// TwinCAT 3 PLC project ExternControl
// ProgramVersion: 3.1.4024.0
// libraries:
//   Tc2_Standard, * (Beckhoff Automation GmbH)
//   Tc2_System, * (Beckhoff Automation GmbH)
//   Tc2_Utilities, * (Beckhoff Automation GmbH)
//   Tc3_Module, * (Beckhoff Automation GmbH)
//   VisuDialogs, * (System)
// project tree:
//   / GlobalTextList.TcGTLO, MAIN.TcPOU, PlcTask.TcTTO
//   MAPPING/ MAP_OUT.TcPOU (not stored), MAP_IN.TcPOU
//   MAPPING/types/ U_MOVER_CTRL.TcDUT (not stored), U_STATION_CTRL.TcDUT, U_STATION_STATE.TcDUT (not stored), U_XTS_TRANSPORT_CTRL.TcDUT, U_XTS_TRANSPORT_STATE.TcDUT (not stored)
//   PROCESS/ fb_Process.TcPOU, GVL_PROCESS.TcGVL (not stored), I_ExternControl_Process.TcIO, PROCESS_CONSTANTS.TcGVL
//   PROCESS/proc/ fb_Worker.TcPOU
//   PROCESS/_types/ E_PROCESS_TYPE.TcDUT
//   PROCESS/_Visualization/ T_PROCESS_VISU.TcVIS, PROCESS_CONTROL.TcVIS (not stored), T_XPU_VISU.TcVIS (not stored), PROCESS_XTS_TRANSPORT.TcVIS
//   XTS_TRANSPORT/CaGroup/types/ E_CA_GROUP_STATE.TcDUT (not stored), E_GROUP_CHECK.TcDUT (not stored), ST_GROUP_INFO.TcDUT
//   XTS_TRANSPORT/ GVL_XTS.TcGVL (not stored), XTS_Parameter.TcGVL
//   XTS_TRANSPORT/Mover/types/ E_MOVER_CTRL.TcDUT, E_MOVER_STATE.TcDUT, ST_GEAR_DATA.TcDUT, ST_MOVER_CTRL.TcDUT (not stored), ST_MOVER_INFO.TcDUT (not stored), ST_MOVER_STATE.TcDUT, ST_MOVE_DATA.TcDUT
//   XTS_TRANSPORT/Xpu/types/ E_XPU_CHECK.TcDUT (not stored), E_XPU_CTRL.TcDUT (not stored), E_XPU_INIT.TcDUT (not stored), E_XPU_STATE.TcDUT, ST_XPU_CTRL.TcDUT (not stored), ST_XPU_INFO.TcDUT, ST_XPU_STATE.TcDUT
//   XTS_TRANSPORT/XtsStation/_types/ E_STATION_CTRL.TcDUT (not stored), E_STATION_STATE.TcDUT (not stored), ST_STATION_CTRL.TcDUT (not stored), ST_STATION_PARAMETER.TcDUT, ST_STATION_STATE.TcDUT
//   XTS_TRANSPORT/XtsTransport/types/ E_XTS_TRANSPORT_CHECK.TcDUT (not stored), E_XTS_TRANSPORT_CTRL.TcDUT, E_XTS_TRANSPORT_STATE.TcDUT, ST_XTS_TRANSPORT_CTRL.TcDUT, ST_XTS_TRANSPORT_STATE.TcDUT (not stored)
//   XTS_TRANSPORT/_types/ E_PROGRESS.TcDUT, f_GetProgress.TcPOU, f_GetState.TcPOU (not stored), f_MoverIdDetectionModeToString.TcPOU (not stored), f_MoverPositionAssignementToString.TcPOU (not stored), f_XpuOperationModeToString.TcPOU (not stored)
//   XTS_TRANSPORT/_Visualization/ GROUP_VISU.TcVIS, STATION_VISU.TcVIS (not stored), Visualization Manager.TcVMO (not stored), XPU_VISU.TcVIS (not stored), XTS_TRANSPORT.TcVIS (not stored)
//   XTS_TRANSPORT/_Visualization/textlists/ TL_E_CTRL_STATION.TcTLO, TL_E_CTRL_TRANSPORT.TcTLO (not stored), TL_E_CTRL_XPU.TcTLO

CONFIGURATION ExternControl
    RESOURCE PLC ON TwinCAT3
        TASK PlcTask(INTERVAL := T#4ms, PRIORITY := 15);
        PROGRAM MAP_IN WITH PlcTask : MAP_IN;
        PROGRAM MAIN WITH PlcTask : MAIN;
        PROGRAM MAP_OUT WITH PlcTask : MAP_OUT;
    END_RESOURCE
END_CONFIGURATION

// ---- MAPPING/types/U_STATION_CTRL.TcDUT
{attribute 'pack_mode' := '2'}
TYPE U_STATION_CTRL :
UNION  
  _st           : ARRAY[1..MAX_STATION] OF ST_STATION_CTRL;
  _by   AT %Q*  : ARRAY[1..MAX_STATION] OF
                  ARRAY[1..SIZEOF(ST_STATION_CTRL)] OF BYTE;
END_UNION
END_TYPE

// ---- MAPPING/types/U_XTS_TRANSPORT_CTRL.TcDUT
{attribute 'pack_mode' := '2'}
TYPE U_XTS_TRANSPORT_CTRL :
UNION
  _st           : ST_XTS_TRANSPORT_CTRL;
  _by   AT%Q*   : ARRAY[1..SIZEOF(ST_XTS_TRANSPORT_CTRL)] OF BYTE;
END_UNION
END_TYPE

// ---- PROCESS/_types/E_PROCESS_TYPE.TcDUT
{attribute 'qualified_only'}
{attribute 'strict'}
{attribute 'to_string'}
TYPE E_PROCESS_TYPE :
(
	NULL,             // nothing happens here
  SINGLE,           // single XTS Station
  PARALLEL,         // synced station handshakes for multiple XTS Stations, same process on all stations, all who enter are processed
  PARALLEL_STRICT,  // synced station handshakes for multiple XTS Stations, same process on all stations, all who are enabled must be processed
  SERIAL,           // synced station handshakes for multiple XTS Stations, all mover have to go through all stations in process
  DISTRIBUTOR       // single XTS Station, no work done here, automated distribution for LastTarget to FirstTarget
)UINT;
END_TYPE

// ---- XTS_TRANSPORT/CaGroup/types/ST_GROUP_INFO.TcDUT
TYPE ST_GROUP_INFO :
STRUCT
  GroupStatusValid,
  GroupStatusBusy,
  GroupMoving, 
  GroupHoming, 
  GroupErrorStop, 
  GroupNotReady, 
  GroupStandby, 
  GroupStopping,
 
  GroupDisabled, 
  AllAxesStanding, 
  ConstantVelocity, 
  Accelerating, 
  Decelerating, 
  InPosition, 
  GroupError					  : BIT; 

  GroupErrorId					: UDINT;

  AxisCount      				: UDINT;
  AxisCountEnabled      : UDINT;

  {attribute 'displaymode':='hex'}
  CaGroupOID            : OTCID;

  CaGroupState          : E_CA_GROUP_STATE;
END_STRUCT
END_TYPE

// ---- XTS_TRANSPORT/Mover/types/E_MOVER_CTRL.TcDUT
{attribute 'qualified_only'}
{attribute 'strict'}
{attribute 'to_string'}
TYPE E_MOVER_CTRL :
(
  MOVER_NULL,               // initial value at startup, used for change of order or retrigger
  MOVER_ENABLE,             // sets MC_Power.Enable
  MOVER_DISABLE,            // removes MC_Power.Enable
  MOVER_MOVE_TO_POS,        // modulo absolute positioning with MC_MoveAbsolute, InTargetPosition check
  MOVER_MOVE_TO_POS_CA,     // modulo absolute positioning with MC_MoveAbsoluteCA, InTargetPosition check
  MOVER_SEND_TO_POS_CA,     // modulo absolute positioning with MC_MoveAbsoluteCA, done after moving ReleaseDistance
  MOVER_HALT,               // halts mover; by use of MC_Halt mover is set passive in CA group
  MOVER_GEAR_IN,            // GearIn for mover in standstill

  MOVER_GEAR_IN_POS_CA,     // GearInPosCA of mover; when FB_GearInPosCa is InSync --> order is done; check SyncDistance yourself and release mover with e_mover_order.mover_SendToPos
  MOVER_GEAR_OUT,           // gear out for mover
  MOVER_RESET               // MC_RESET for mover
)UINT;
END_TYPE

// ---- XTS_TRANSPORT/Mover/types/E_MOVER_STATE.TcDUT
{attribute 'qualified_only'}
{attribute 'to_string'}
TYPE E_MOVER_STATE :
(
  MOVER_NULL,               // initial value at startup, used for change of order or retrigger
  MOVER_ENABLE,             // sets MC_Power.Enable
  MOVER_DISABLE,            // removes MC_Power.Enable
  MOVER_MOVE_TO_POS,        // modulo absolute positioning with MC_MoveAbsolute, InTargetPosition check
  MOVER_MOVE_TO_POS_CA,     // modulo absolute positioning with MC_MoveAbsoluteCA, InTargetPosition check
  MOVER_SEND_TO_POS_CA,     // modulo absolute positioning with MC_MoveAbsoluteCA, done after moving ReleaseDistance
  MOVER_HALT,               // halts mover; by use of MC_Halt mover is set passive in CA group
  MOVER_GEAR_IN,            // GearIn for mover in standstill

  MOVER_GEAR_IN_POS_CA,     // GearInPosCA of mover; when FB_GearInPosCa is InSync --> order is done; check SyncDistance yourself and release mover with e_mover_order.mover_SendToPos
  MOVER_GEAR_OUT,           // gear out for mover
  MOVER_RESET               // MC_RESET for mover
)UINT;
END_TYPE

// ---- XTS_TRANSPORT/Mover/types/ST_GEAR_DATA.TcDUT
{attribute 'pack_mode' := '2'}
TYPE ST_GEAR_DATA :
STRUCT
  rDeltaToMasterPos       : REAL;
  rModuloSyncPosSlave     : REAL;
  rMasterStartDistance    : REAL;
  rGearNumerator          : REAL;
  iGearDenumerator        : USINT  := 1;
END_STRUCT
END_TYPE

// ---- XTS_TRANSPORT/Mover/types/ST_MOVER_STATE.TcDUT
{attribute 'pack_mode' := '2'}
TYPE ST_MOVER_STATE :
STRUCT
  State           : E_MOVER_STATE;  // ST_MOVER_CTRL.Cmd with added E_PROGRESS
  MasterId        : USINT;            // mirror NC AxisId of Master axis
END_STRUCT
END_TYPE

// ---- XTS_TRANSPORT/Mover/types/ST_MOVE_DATA.TcDUT
{attribute 'pack_mode' := '2'}
TYPE ST_MOVE_DATA :
STRUCT
  // HAUD 2024 03 14
  // some init data added for example
  rPos            : LREAL :=   2275.0;
  rVelo           : LREAL :=    500.0;
  rAcc            : LREAL :=   5000.0;
  rJerk           : LREAL := 500000.0;
  rGap            : LREAL :=    100.0;
  rOverride       : LREAL :=    100.0;
  rDelta          : LREAL :=      0.05;
  rDistance       : LREAL :=     25.0;
END_STRUCT
END_TYPE

// ---- XTS_TRANSPORT/Xpu/types/E_XPU_STATE.TcDUT
{attribute 'to_string'}
TYPE E_XPU_STATE :
(
  XTS_NULL,
  XTS_INVALID,
  XTS_INIT                      := 10,    // initialize XPU
  XTS_STATION_INFO_READ         := 20,    // get Station information from Xpu
  XTS_IDLE                      := 30
)UINT;
END_TYPE

// ---- XTS_TRANSPORT/Xpu/types/ST_XPU_INFO.TcDUT
{attribute 'pack_mode' := '2'}
TYPE ST_XPU_INFO :
STRUCT
  AllPositionsValid   : BIT;
  IdDetectionError    : BIT;
  IdDetectionValid    : BIT;
  IdDetectionActive   : BIT;

  OperationMode       : UINT;

  IdDetectionMode           : UINT;
  MoverPositionAssignement  : UINT;

  nDetectedAxisCount  : UINT;
  nExpectedAxisCount  : UINT;

  
END_STRUCT
END_TYPE

// ---- XTS_TRANSPORT/Xpu/types/ST_XPU_STATE.TcDUT
{attribute 'pack_mode' := '2'}
TYPE ST_XPU_STATE :
STRUCT
  Init            : E_XPU_INIT;
  State           : E_XPU_STATE;
  Check           : E_XPU_CHECK;
  DcLink          : BIT;
END_STRUCT
END_TYPE

// ---- XTS_TRANSPORT/XtsStation/_types/ST_STATION_PARAMETER.TcDUT
TYPE ST_STATION_PARAMETER :
STRUCT
  sText             : STRING(80); // only description
  rPosWait          : REAL;       // start of station, a sending station is using this value to send mover to
  rReleaseDistance  : REAL;       // distance from stop pos mover has to travel (from ActPos) in order for station to go back to mover detection

  rGap              : REAL;
  rVelo             : REAL;
  rAccDec           : REAL;
  rJerk             : REAL;

  // how many nests (stop positions) mover has to stop at (1 = default)
  nConfiguredStopCount  : USINT := 1; // 1-8 --> NestMask = BYTE

  // mover stop position in station, relative to rPosWait!!
  rPosStop          : ARRAY[1..8] OF LREAL;
END_STRUCT
END_TYPE

// ---- XTS_TRANSPORT/XtsStation/_types/ST_STATION_STATE.TcDUT
{attribute 'pack_mode' := '2'}
TYPE ST_STATION_STATE :
STRUCT
  eState          : E_STATION_STATE;
  {attribute 'displaymode':='bin'}
  nMask           : BYTE;
  nMoverId        : USINT;
  rMoverModPos    : lreal; // modulo position of detected mover
  nQueue          : USINT; // queue count for station
END_STRUCT
END_TYPE

// ---- XTS_TRANSPORT/XtsTransport/types/E_XTS_TRANSPORT_CTRL.TcDUT
{attribute 'strict'}
{attribute 'to_string'}
TYPE E_XTS_TRANSPORT_CTRL :
(
  CMD_NULL,
  CMD_INIT                  := 10,  // Xpu, Group, Mover initialization: clear errors, clear group, check Xpu data, check mover detection
  CMD_IDLE,

  CMD_MOVER_ENABLE          := 20,  // all mover are enabled, checked for ControlLoopClosed
  CMD_MOVER_DISABLE,                // all mover are disabled, no axis in CaGroup: no error, any axis in CaGroup: group error

  CMD_GROUP_CLEAR           := 30,  // halt all movers, clear errors, remove all movers from group, clear group
  CMD_GROUP_BUILD,                  // add all movers to group
  CMD_GROUP_ENABLE,                 // group with movers is enabled

  CMD_TRANSPORT_START       := 40,  // move all mover[i] to start position
  CMD_TRANSPORT_RESTART             // move all mover[i] to LastPosition[i]

)UINT;
END_TYPE

// ---- XTS_TRANSPORT/XtsTransport/types/E_XTS_TRANSPORT_STATE.TcDUT
{attribute 'to_string'}
TYPE E_XTS_TRANSPORT_STATE :
(
  TRANSPORT_NULL,
  TRANSPORT_INVALID,
  TRANSPORT_INIT            := 10,  // Xpu, Group, Mover initialization: init TcCOM objects, clear errors, clear group, check Xpu data, check mover detection
  TRANSPORT_IDLE,                   // cyclic check for errors, check Xpu data

  TRANSPORT_MOVER_ENABLE    := 20,  // all mover are enabled, checked for ControlLoopClosed
  TRANSPORT_MOVER_DISABLE,          // all mover are disabled

  TRANSPORT_GROUP_CLEAR     := 30,  // halt all movers, clear errors, remove all movers from group, clear group
  TRANSPORT_GROUP_BUILD,            // add all movers to group
  TRANSPORT_GROUP_ENABLE,           // group with movers is enabled

  TRANSPORT_START           := 40,  // move all mover[i] to start position
  TRANSPORT_RESTART                 // move all mover[i] to LastPosition[i]
)UINT;
END_TYPE

// ---- XTS_TRANSPORT/XtsTransport/types/ST_XTS_TRANSPORT_CTRL.TcDUT
TYPE ST_XTS_TRANSPORT_CTRL :
STRUCT
  Cmd       : E_XTS_TRANSPORT_CTRL;
END_STRUCT
END_TYPE

// ---- XTS_TRANSPORT/_types/E_PROGRESS.TcDUT
{attribute 'qualified_only'}
{attribute 'to_string'}
TYPE E_PROGRESS :
(
  PROGRESS_INVALID,
  PROGRESS_INIT           :=  1000,
  PROGRESS_BUSY           :=  2000,
  PROGRESS_PREPARE        :=  3000,
  PROGRESS_STARTUP        :=  4000,
  PROGRESS_CHECK          :=  5000,
  PROGRESS_OCCUPIED       :=  6000,
  PROGRESS_WORKING        :=  7000,
  PROGRESS_STILL_WORKING  :=  8000,
  PROGRESS_ERROR          :=  9000,
  PROGRESS_DONE           := 10000
)UINT;
END_TYPE

// ---- PROCESS/PROCESS_CONSTANTS.TcGVL
//{attribute 'qualified_only'}
VAR_GLOBAL CONSTANT
  MAX_PROCESS       : UINT := 9;

  DISTRIBUTOR_2     : UINT := 9;// 9
  DISTRIBUTOR_1     : UINT := 8;// 8
  OUTPUT_R2         : UINT := 7;// 7
  OUTPUT_R1         : UINT := 6;// 6
  BUFFER_3          : UINT := 5;// 5
  OUTPUT_1          : UINT := 4;// 4
  INPUT             : UINT := 3;// 3
  BUFFER_1          : UINT := 2;// 2
  BUFFER_4          : UINT := 1;// 1

  QUEUE_COUNT       : UINT := 12; // 
END_VAR

// ---- XTS_TRANSPORT/XTS_Parameter.TcGVL
//{attribute 'qualified_only'}
VAR_GLOBAL CONSTANT
// HAUD 2024 04 30 - introduction of fb_UnitControl
  Version             : STRING  := '3.2.8';

  MAX_MOVER           : UINT    := 96;

  MAX_STATION         : UINT    := 53;
  MAX_STATION_NEST    : UINT    := TO_UINT(SIZEOF(ST_STATION_STATE.nMask)*8);

END_VAR

// ---- PROCESS/I_ExternControl_Process.TcIO
INTERFACE I_ExternControl_Process

METHOD PUBLIC DelBitWord : WORD
VAR_INPUT
  inVal   : WORD;
  bitNo   : DINT;
END_VAR
END_METHOD

PROPERTY EnableProcess : word
GET
END_GET
SET
END_SET
END_PROPERTY

METHOD PUBLIC GetBitDWord : BOOL
VAR_INPUT
  inVal   : DWORD;
  bitNo   : DINT;
END_VAR
END_METHOD

METHOD PUBLIC GetBitWord : BOOL
VAR_INPUT
  inVal   : WORD;
  bitNo   : DINT;
END_VAR
END_METHOD

METHOD PUBLIC Init : BOOL
END_METHOD

PROPERTY MoverCountInQueue : uint
GET
END_GET
END_PROPERTY

PROPERTY MoverInQueue : Bool
GET
END_GET
END_PROPERTY

PROPERTY ProcessCmd : E_STATION_CTRL
SET
END_SET
END_PROPERTY

PROPERTY ProcessPerMinute : uint
GET
END_GET
END_PROPERTY

PROPERTY ProcessState : E_STATION_STATE
GET
END_GET
END_PROPERTY

PROPERTY ProcessType : e_process_type
GET
END_GET
SET
END_SET
END_PROPERTY

METHOD PUBLIC SetBitDWord : DWORD
VAR_INPUT
  inVal   : DWORD;
  bitNo   : DINT;
END_VAR
END_METHOD

METHOD PUBLIC SetBitWord : WORD
VAR_INPUT
  inVal   : WORD;
  bitNo   : DINT;
END_VAR
END_METHOD

PROPERTY StationCount : uint
GET
END_GET
END_PROPERTY

PROPERTY StationFirst : uint
GET
END_GET
SET
END_SET
END_PROPERTY

PROPERTY TargetMask : dword
GET
END_GET
SET
END_SET
END_PROPERTY

END_INTERFACE

// ---- MAPPING/MAP_IN.TcPOU
PROGRAM MAP_IN
VAR

  {attribute 'TcLinkTo' := '._by := TIPC^XtsTransport^XtsTransport Instance^PlcTask Outputs^MAP_OUT.uTransportState._by'}
  uTransportState     : U_XTS_TRANSPORT_STATE;
  {attribute 'TcLinkTo' := '._by := TIPC^XtsTransport^XtsTransport Instance^PlcTask Outputs^MAP_OUT.uStationState._by'}
  uStationState       : U_STATION_STATE;
END_VAR

          // destination address
                                            // source address
                                                                    // size
  memcpy(ADR(GVL_XTS.XtsTransportState),  ADR(uTransportState),   SIZEOF(ST_XTS_TRANSPORT_STATE));
  memcpy(ADR(GVL_XTS.StationState),       ADR(uStationState),     SIZEOF(uStationState));

END_PROGRAM

// ---- MAIN.TcPOU
//---------------------------------------------------------------------------------------------------------------
//
//  HAUD 2024.04.13
//
//  - ExternControl for XtsTransport
//
//  - example project for controlling XTS transport layer
//  - transport layer members:
//
//      HAUD 2024 04 30 - introduction of fb_UnitControl as interface to APPLICATION
//
//    - fb_UnitControl
//      - groups commands into sequences for APPLICATION
//      - handles XtsTransport
//      - handles fb_Process
//
//    - fb_Process
//      - groups XtsStations for processes
//      - synced handshakes with all assigned XtsStations
//
//    - Transport Control Unit
//      - mapped from XtsTransport GVL_XTS.TransportCtrl / GVL_XTS.TransportState
//        - Info for CaGroup
//        - Info for Xpu
//
//      - coordinates members to get XTS in defined states
//
//    - Xts Stations
//      - handshakes for mover transport
//
//---------------------------------------------------------------------------------------------------------------
// This SOFTWARE is provided as an Exemple by THE PROVIDER "as is" and "with all faults." THE PROVIDER makes no 
// representations or warranties of any kind concerning the safety, suitability, lack of viruses, inaccuracies, 
// typographical errors, or other harmful components of this SOFTWARE. There are inherent dangers in the use of 
// any software, and you are solely responsible for determining whether this SOFTWARE is compatible with your 
// equipment and other software installed on your equipment. You are also solely responsible for the protection 
// of your equipment and backup of your data, and THE PROVIDER will not be liable for any damages you may suffer 
// in connection with using, modifying, or distributing this SOFTWARE.
//---------------------------------------------------------------------------------------------------------------
PROGRAM MAIN
VAR
  bInit,
  bStart              : BOOL;
  eInit               : E_PROGRESS;

  nProcess,
  nStation            : UINT;

  tProcess            : ARRAY[1..MAX_PROCESS] OF TIME;

  {attribute 'displaymode':='bin'}
  wEnableProcess      : ARRAY[1..MAX_PROCESS] OF DWORD;  // switch XTS stations on/off here (one word per process --> max. 16 stations each)

  {attribute 'displaymode':='bin'}
  wInitProcess        : WORD;  // processes init

  bEmptySerialStation : BOOL;

  eProcessCmd         : ARRAY[1..MAX_PROCESS] OF E_STATION_CTRL;
  eProcessState       : ARRAY[1..MAX_PROCESS] OF E_STATION_STATE;

  nMoverSelected,
  nStationSelected,
  nProcessSelected,
  nStationParameter   : UINT;

  eTransportCmd,
  eTransportCmdOld    : E_XTS_TRANSPORT_CTRL;

  eTransportState,
  eTransportStateOld  : E_XTS_TRANSPORT_STATE;
  eTransportResult,
  eStateStart         : E_PROGRESS;

  eXpuState           : E_XPU_STATE;
  eXpuResult          : E_PROGRESS;
  eXpuCheck           : E_XPU_CHECK;

  eMoverState         : E_MOVER_STATE;
  eMoverResult        : E_PROGRESS;

  sCaGroupState,
  sTransportState,
  sTransportCheck,
  sTransportResult,
  sXpuState,
  sXpuResult,
  sXpuCheck,
  sXpuOpMode,
  sXpuMoverdetectionMode,
  sXpuMoverAssignement,
  sMoverState,
  sMoverResult,
  sStationState,
  sStationStateMask,
  sStationCtrlMask,
  sProcessEnableMask        : STRING;

  bStationEnable,
  bStationEnter,
  bStationStart,
  bStationDone,
  bStationOut,
  bStationGone            : BOOL;

  sStationText            : STRING;
  nVariant                : uint;
END_VAR

//#############################################################################
// Visualization data	
//#############################################################################	
VisuData();
//
//#############################################################################
// check for changed Cmd on XtsTransportCtrl.Cmd
//#############################################################################
//
eTransportCmd                         := GVL_XTS.XtsTransportCtrl.Cmd;
//
IF (eTransportCmd <> eTransportCmdOld)
THEN
  eTransportCmdOld                    := eTransportCmd;
  bStart                              := FALSE;
  bEmptySerialStation                 := FALSE;
  eStateStart                         := E_PROGRESS.PROGRESS_INIT;
  memset(ADR(wEnableProcess), 0, SIZEOF(wEnableProcess));

  CASE eTransportCmd
  OF
    E_XTS_TRANSPORT_CTRL.CMD_INIT:
      bInit                           := FALSE;

  ELSE
    IF bInit
    THEN
      CASE eTransportCmd
      OF
        E_XTS_TRANSPORT_CTRL.CMD_IDLE,
        E_XTS_TRANSPORT_CTRL.CMD_TRANSPORT_START:
          FOR nProcess := 1 TO MAX_PROCESS
          DO
            eProcessCmd[nProcess]     := E_STATION_CTRL.STATION_DISABLE;
          END_FOR
      END_CASE
    END_IF
  END_CASE
END_IF
//
//
//#############################################################################
// check for changed state on XtsTransportState.State
//#############################################################################
//
IF (GVL_XTS.XtsTransportState.State <> eTransportStateOld)
THEN
  CASE (GVL_XTS.XtsTransportState.State MOD E_PROGRESS.PROGRESS_DONE)
  OF
    E_XTS_TRANSPORT_STATE.TRANSPORT_START:
      CASE eStateStart
      OF
        E_PROGRESS.PROGRESS_INIT:
          IF GVL_XTS.XtsTransportState.GroupInfo.AllAxesStanding
          THEN
            eStateStart               := E_PROGRESS.PROGRESS_BUSY;
            memset(ADR(wEnableProcess), 0, SIZEOF(wEnableProcess));
          END_IF

        E_PROGRESS.PROGRESS_BUSY:
          eStateStart                   := E_PROGRESS.PROGRESS_PREPARE;
          FOR nProcess := 1 TO MAX_PROCESS
          DO
            FOR nStation := 1 TO GVL_PROCESS.Process[nProcess].StationCount
            DO
              wEnableProcess[nProcess]  := GVL_PROCESS.Process[nProcess].SetBitDWord(wEnableProcess[nProcess],(nStation-1));
            END_FOR
            //wEnableProcess[OUTPUT_R1] := 1;
            GVL_PROCESS.Process[nProcess].EnableProcess := TO_WORD(wEnableProcess[nProcess]);
          END_FOR
          FOR nProcess := 1 TO MAX_PROCESS
          DO
            IF (nProcess = MAX_PROCESS)
            THEN
              GVL_PROCESS.Process[nProcess].TargetMask := wEnableProcess[1];
            ELSE
              GVL_PROCESS.Process[nProcess].TargetMask := wEnableProcess[nProcess+1];
            END_IF
          END_FOR
          FOR nStation := 0 TO (GVL_PROCESS.Process[BUFFER_3].TargetLast - GVL_PROCESS.Process[BUFFER_3].TargetFirst)
          DO 
            GVL_PROCESS.Process[BUFFER_3].TargetMask     := GVL_PROCESS.Process[BUFFER_3].SetBitDWord(GVL_PROCESS.Process[BUFFER_3].TargetMask,(nStation));
          END_FOR

        E_PROGRESS.PROGRESS_PREPARE:
          eStateStart                 := E_PROGRESS.PROGRESS_STARTUP;
          FOR nProcess := 1 TO MAX_PROCESS
          DO
            IF NOT (GVL_PROCESS.Process[nProcess].EnableProcess = wEnableProcess[nProcess])
            THEN
              eStateStart             := E_PROGRESS.PROGRESS_PREPARE;
            END_IF
          END_FOR

        E_PROGRESS.PROGRESS_STARTUP:
          eTransportStateOld          := GVL_XTS.XtsTransportState.State;
          bStart                      := TRUE;
      END_CASE

  ELSE
    eTransportStateOld                := GVL_XTS.XtsTransportState.State;

    CASE (GVL_XTS.XtsTransportState.State MOD E_PROGRESS.PROGRESS_ERROR)
    OF
      E_XTS_TRANSPORT_STATE.TRANSPORT_START:
        bStart                        := FALSE;

    END_CASE
  END_CASE
END_IF
//
//#############################################################################
//#############################################################################
//
IF NOT bInit
THEN
  Init();
  ProcessConfig_2x12_DST_02();
END_IF
//#############################################################################
//#############################################################################
// cyclic call to processes
//#############################################################################
FOR nProcess := 1 TO MAX_PROCESS
DO
  GVL_PROCESS.Process[nProcess].Cycle();

  GVL_PROCESS.Process[nProcess].EnabledStation    := ADR(GVL_PROCESS.StationsEnabled);  // enabled process: for other processes to read
  GVL_PROCESS.Process[nProcess].MoverPerMinute    := ADR(GVL_PROCESS.MoverPerMinute);

  GVL_PROCESS.Process[nProcess].StationCtrl       := ADR(GVL_XTS.StationCtrl);
  GVL_PROCESS.Process[nProcess].StationState      := ADR(GVL_XTS.StationState);

  GVL_PROCESS.ItfProcess[nProcess]                := GVL_PROCESS.Process[nProcess]; 
END_FOR


//#############################################################################
// process workers
//#############################################################################
GVL_PROCESS.Distributor2.ProcessTime    := tProcess[DISTRIBUTOR_2];
GVL_PROCESS.Distributor2.ProcessIndex   := DISTRIBUTOR_2;
GVL_PROCESS.Distributor2.ItfProcesses   REF= GVL_PROCESS.ItfProcess;

GVL_PROCESS.Distributor1.ProcessTime    := tProcess[DISTRIBUTOR_1];
GVL_PROCESS.Distributor1.ProcessIndex   := DISTRIBUTOR_1;
GVL_PROCESS.Distributor1.ItfProcesses   REF= GVL_PROCESS.ItfProcess;

GVL_PROCESS.OutputR2.ProcessTime        := tProcess[OUTPUT_R2];
GVL_PROCESS.OutputR2.ProcessIndex       := OUTPUT_R2;
GVL_PROCESS.OutputR2.ItfProcesses       REF= GVL_PROCESS.ItfProcess;

GVL_PROCESS.OutputR1.ProcessTime        := tProcess[OUTPUT_R1];
GVL_PROCESS.OutputR1.ProcessIndex       := OUTPUT_R1;
GVL_PROCESS.OutputR1.ItfProcesses       REF= GVL_PROCESS.ItfProcess;

GVL_PROCESS.Buffer3.ProcessTime         := tProcess[BUFFER_3];
GVL_PROCESS.Buffer3.ProcessIndex        := BUFFER_3;
GVL_PROCESS.Buffer3.ItfProcesses        REF= GVL_PROCESS.ItfProcess;

GVL_PROCESS.Output1.ProcessTime         := tProcess[OUTPUT_1];
GVL_PROCESS.Output1.ProcessIndex        := OUTPUT_1;
GVL_PROCESS.Output1.ItfProcesses        REF= GVL_PROCESS.ItfProcess;

GVL_PROCESS.Input1.ProcessTime          := tProcess[INPUT];
GVL_PROCESS.Input1.ProcessIndex         := INPUT;
GVL_PROCESS.Input1.ItfProcesses         REF= GVL_PROCESS.ItfProcess;

GVL_PROCESS.Buffer1.ProcessTime         := tProcess[BUFFER_1];
GVL_PROCESS.Buffer1.ProcessIndex        := BUFFER_1;
GVL_PROCESS.Buffer1.ItfProcesses        REF= GVL_PROCESS.ItfProcess;

GVL_PROCESS.Buffer1.ProcessTime         := tProcess[BUFFER_1];
GVL_PROCESS.Buffer4.ProcessIndex        := BUFFER_4;
GVL_PROCESS.Buffer4.ItfProcesses        REF= GVL_PROCESS.ItfProcess;

//#############################################################################
//
IF NOT (bInit) THEN RETURN; END_IF
//
//#############################################################################
//#############################################################################

IF (nVariant = 0)
THEN
  GVL_PROCESS.Distributor2.AUTO(bStart);
  GVL_PROCESS.Distributor1.AUTO(bStart);
  GVL_PROCESS.OutputR2.AUTO(bStart);
  GVL_PROCESS.OutputR1.AUTO(bStart);
  GVL_PROCESS.Buffer3.AUTO(bStart);
  GVL_PROCESS.Output1.AUTO(bStart);
  GVL_PROCESS.Input1.AUTO(bStart);
  GVL_PROCESS.Buffer1.AUTO(bStart);
  GVL_PROCESS.Buffer4.AUTO(bStart);

ELSIF (nVariant = 1)
THEN
  GVL_PROCESS.Distributor2.AUTO_1(bStart);
  GVL_PROCESS.Distributor1.AUTO_1(bStart);
  GVL_PROCESS.OutputR2.AUTO_1(bStart);
  GVL_PROCESS.OutputR1.AUTO_1(bStart);
  GVL_PROCESS.Buffer3.AUTO_1(bStart);
  GVL_PROCESS.Output1.AUTO_1(bStart);
  GVL_PROCESS.Input1.AUTO_1(bStart);
  GVL_PROCESS.Buffer1.AUTO_1(bStart);
  GVL_PROCESS.Buffer4.AUTO_1(bStart);
END_IF















//#############################################################################

METHOD Init
VAR_INPUT
END_VAR
CASE eInit
OF
  E_PROGRESS.PROGRESS_INVALID,
  E_PROGRESS.PROGRESS_DONE:
    bStart                          := FALSE;
    eInit                           := E_PROGRESS.PROGRESS_INIT;
    GVL_XTS.XtsTransportCtrl.Cmd    := E_XTS_TRANSPORT_CTRL.CMD_NULL;

  E_PROGRESS.PROGRESS_INIT:
    IF (GVL_XTS.XtsTransportState.XpuInfo.IdDetectionValid) OR
       (GVL_XTS.XtsTransportState.XpuInfo.OperationMode = 1) // Simulation
    THEN
      GVL_XTS.XtsTransportCtrl.Cmd  := E_XTS_TRANSPORT_CTRL.CMD_INIT;

      IF (GVL_xts.XtsTransportState.State = E_XTS_TRANSPORT_STATE.TRANSPORT_INIT + E_PROGRESS.PROGRESS_DONE)
      THEN
        GVL_XTS.XtsTransportCtrl.Cmd:= E_XTS_TRANSPORT_CTRL.CMD_IDLE;
        eInit                       := E_PROGRESS.PROGRESS_BUSY;
      END_IF
    END_IF

  E_PROGRESS.PROGRESS_BUSY:
    eInit                           := E_PROGRESS.PROGRESS_PREPARE;
    wInitProcess                    := 0;
    ProcessConfig_1x12();
    ProcessConfig_2x12();

  E_PROGRESS.PROGRESS_PREPARE:
    ProcessConfig_2x12_DST_02();

    FOR nProcess := 1 TO MAX_PROCESS
    DO
      GVL_PROCESS.Process[nProcess].ProcessCmd         := E_STATION_CTRL.STATION_INIT;
      IF (GVL_PROCESS.Process[nProcess].ProcessState = E_STATION_STATE.STATION_INIT)
      THEN
        wInitProcess                := GVL_PROCESS.Process[nProcess].SetBitWord(wInitProcess,  (nProcess-1));
      END_IF
    END_FOR
    IF (wInitProcess = EXPT(2,MAX_PROCESS)-1)
    THEN
      eInit                         := E_PROGRESS.PROGRESS_STARTUP;
    END_IF

  E_PROGRESS.PROGRESS_STARTUP:
    StationParameterInit();

    tProcess[INPUT]                 := T#450MS;
    tProcess[OUTPUT_1]              := T#600MS;
    tProcess[OUTPUT_R1]             := T#600MS;
    tProcess[OUTPUT_R2]             := T#600MS;

    FOR nProcess := 1 TO MAX_PROCESS
    DO
      GVL_PROCESS.Process[nProcess].ProcessCmd         := E_STATION_CTRL.STATION_DISABLE;
    END_FOR
    bInit                           := TRUE;
    eInit                           := E_PROGRESS.PROGRESS_DONE;

END_CASE
END_METHOD

METHOD ProcessConfig_1x12
VAR
  _nProcess     : UINT;
END_VAR

      // BUFFER_4
      _nProcess                       := 1;
      GVL_PROCESS.Process[_nProcess].ProcessType   := E_PROCESS_TYPE.DISTRIBUTOR;
      GVL_PROCESS.Process[_nProcess].StationFirst  := 52;
      GVL_PROCESS.Process[_nProcess].StationLast   := 52;
      GVL_PROCESS.Process[_nProcess].TargetFirst   := 53;
      GVL_PROCESS.Process[_nProcess].TargetLast    := 53;

      // BUFFER_1
      _nProcess                       := 2;
      GVL_PROCESS.Process[_nProcess].ProcessType   := E_PROCESS_TYPE.DISTRIBUTOR;
      GVL_PROCESS.Process[_nProcess].StationFirst  := 53;
      GVL_PROCESS.Process[_nProcess].StationLast   := 53;
      GVL_PROCESS.Process[_nProcess].TargetFirst   :=  1;
      GVL_PROCESS.Process[_nProcess].TargetLast    := 12;

      // INPUT
      _nProcess                       := 3;
      tProcess[_nProcess]             := T#850MS;
      GVL_PROCESS.Process[_nProcess].ProcessType   := E_PROCESS_TYPE.PARALLEL;
      GVL_PROCESS.Process[_nProcess].StationFirst  :=  1;
      GVL_PROCESS.Process[_nProcess].StationLast   := 12;
      GVL_PROCESS.Process[_nProcess].TargetFirst   := 13;
      GVL_PROCESS.Process[_nProcess].TargetLast    := 24;

      // OUTPUT_1
      _nProcess                       := 4;
      tProcess[_nProcess]             := T#850MS;
      GVL_PROCESS.Process[_nProcess].ProcessType   := E_PROCESS_TYPE.PARALLEL;
      GVL_PROCESS.Process[_nProcess].StationFirst  := 13;
      GVL_PROCESS.Process[_nProcess].StationLast   := 24;
      GVL_PROCESS.Process[_nProcess].TargetFirst   := 50;
      GVL_PROCESS.Process[_nProcess].TargetLast    := 50;

      // DISTRIBUTOR_1
      _nProcess                        := 8;
      GVL_PROCESS.Process[_nProcess].ProcessType   := E_PROCESS_TYPE.DISTRIBUTOR;
      GVL_PROCESS.Process[_nProcess].StationFirst  := 50;
      GVL_PROCESS.Process[_nProcess].StationLast   := 50;
      GVL_PROCESS.Process[_nProcess].TargetFirst   := 51;
      GVL_PROCESS.Process[_nProcess].TargetLast    := 51;

      // DISTRIBUTOR_2
      _nProcess                        := 9;
      GVL_PROCESS.Process[_nProcess].ProcessType   := E_PROCESS_TYPE.DISTRIBUTOR;
      GVL_PROCESS.Process[_nProcess].StationFirst  := 51;
      GVL_PROCESS.Process[_nProcess].StationLast   := 51;
      GVL_PROCESS.Process[_nProcess].TargetFirst   := 52;
      GVL_PROCESS.Process[_nProcess].TargetLast    := 52;
END_METHOD

METHOD ProcessConfig_2x12
VAR
  _nProcess     : UINT;
END_VAR
    
      // BUFFER_4
      _nProcess                       := BUFFER_4;
      GVL_PROCESS.Process[_nProcess].ProcessType   := E_PROCESS_TYPE.DISTRIBUTOR;
      GVL_PROCESS.Process[_nProcess].StationFirst  := 52;
      GVL_PROCESS.Process[_nProcess].StationLast   := 52;
      GVL_PROCESS.Process[_nProcess].TargetFirst   := 53;
      GVL_PROCESS.Process[_nProcess].TargetLast    := 53;

      // BUFFER_1
      _nProcess                       := BUFFER_1;
      GVL_PROCESS.Process[_nProcess].ProcessType   := E_PROCESS_TYPE.DISTRIBUTOR;
      GVL_PROCESS.Process[_nProcess].StationFirst  := 53;
      GVL_PROCESS.Process[_nProcess].StationLast   := 53;
      GVL_PROCESS.Process[_nProcess].TargetFirst   :=  1;
      GVL_PROCESS.Process[_nProcess].TargetLast    := 12;

      // INPUT
      _nProcess                       := INPUT;
      GVL_PROCESS.Process[_nProcess].ProcessType   := E_PROCESS_TYPE.PARALLEL;
      GVL_PROCESS.Process[_nProcess].StationFirst  :=  1;
      GVL_PROCESS.Process[_nProcess].StationLast   := 12;
      GVL_PROCESS.Process[_nProcess].TargetFirst   := 25;
      GVL_PROCESS.Process[_nProcess].TargetLast    := 25;

      // BUFFER_3
      _nProcess                        := BUFFER_3;
      GVL_PROCESS.Process[_nProcess].ProcessType   := E_PROCESS_TYPE.DISTRIBUTOR;
      GVL_PROCESS.Process[_nProcess].StationFirst  := 25;
      GVL_PROCESS.Process[_nProcess].StationLast   := 25;
      GVL_PROCESS.Process[_nProcess].TargetFirst   := 26;
      GVL_PROCESS.Process[_nProcess].TargetLast    := 49;

      // OUTPUT_R1
      _nProcess                        := OUTPUT_R1;
      GVL_PROCESS.Process[_nProcess].ProcessType   := E_PROCESS_TYPE.PARALLEL_STRICT;
      GVL_PROCESS.Process[_nProcess].StationFirst  := 26;
      GVL_PROCESS.Process[_nProcess].StationLast   := 37;
      GVL_PROCESS.Process[_nProcess].TargetFirst   := 50;
      GVL_PROCESS.Process[_nProcess].TargetLast    := 50;

      // OUTPUT_R2
      _nProcess                        := OUTPUT_R2;
      GVL_PROCESS.Process[_nProcess].ProcessType   := E_PROCESS_TYPE.PARALLEL_STRICT;
      GVL_PROCESS.Process[_nProcess].StationFirst  := 38;
      GVL_PROCESS.Process[_nProcess].StationLast   := 49;
      GVL_PROCESS.Process[_nProcess].TargetFirst   := 50;
      GVL_PROCESS.Process[_nProcess].TargetLast    := 50;

      // DISTRIBUTOR_1
      _nProcess                        := DISTRIBUTOR_1;
      GVL_PROCESS.Process[_nProcess].ProcessType   := E_PROCESS_TYPE.DISTRIBUTOR;
      GVL_PROCESS.Process[_nProcess].StationFirst  := 50;
      GVL_PROCESS.Process[_nProcess].StationLast   := 50;
      GVL_PROCESS.Process[_nProcess].TargetFirst   := 51;
      GVL_PROCESS.Process[_nProcess].TargetLast    := 51;

      // DISTRIBUTOR_2
      _nProcess                        := DISTRIBUTOR_2;
      GVL_PROCESS.Process[_nProcess].ProcessType   := E_PROCESS_TYPE.DISTRIBUTOR;
      GVL_PROCESS.Process[_nProcess].StationFirst  := 51;
      GVL_PROCESS.Process[_nProcess].StationLast   := 51;
      GVL_PROCESS.Process[_nProcess].TargetFirst   := 52;
      GVL_PROCESS.Process[_nProcess].TargetLast    := 52;
END_METHOD

METHOD ProcessConfig_2x12_DST_02
VAR
  _nProcess     : UINT;
END_VAR
    
      // BUFFER_4
      _nProcess                       := BUFFER_4;
      GVL_PROCESS.Process[_nProcess].ProcessType   := E_PROCESS_TYPE.DISTRIBUTOR;
      GVL_PROCESS.Process[_nProcess].StationFirst  := 52;
      GVL_PROCESS.Process[_nProcess].StationLast   := 52;
      GVL_PROCESS.Process[_nProcess].TargetFirst   := 53;
      GVL_PROCESS.Process[_nProcess].TargetLast    := 53;

      // BUFFER_1
      _nProcess                       := BUFFER_1;
      GVL_PROCESS.Process[_nProcess].ProcessType   := E_PROCESS_TYPE.DISTRIBUTOR;
      GVL_PROCESS.Process[_nProcess].StationFirst  := 53;
      GVL_PROCESS.Process[_nProcess].StationLast   := 53;
      GVL_PROCESS.Process[_nProcess].TargetFirst   :=  1;
      GVL_PROCESS.Process[_nProcess].TargetLast    := 12;

      // INPUT
      _nProcess                       := INPUT;
      GVL_PROCESS.Process[_nProcess].ProcessType   := E_PROCESS_TYPE.PARALLEL;
      GVL_PROCESS.Process[_nProcess].StationFirst  :=  1;
      GVL_PROCESS.Process[_nProcess].StationLast   := 12;
      GVL_PROCESS.Process[_nProcess].TargetFirst   := 25;
      GVL_PROCESS.Process[_nProcess].TargetLast    := 25;

      // BUFFER_3
      _nProcess                        := BUFFER_3;
      GVL_PROCESS.Process[_nProcess].ProcessType   := E_PROCESS_TYPE.DISTRIBUTOR;
      GVL_PROCESS.Process[_nProcess].StationFirst  := 25;
      GVL_PROCESS.Process[_nProcess].StationLast   := 25;
      GVL_PROCESS.Process[_nProcess].TargetFirst   := 26;
      GVL_PROCESS.Process[_nProcess].TargetLast    := 49;

      // OUTPUT_R1
      _nProcess                        := OUTPUT_R1;
      GVL_PROCESS.Process[_nProcess].ProcessType   := E_PROCESS_TYPE.PARALLEL_STRICT;
      GVL_PROCESS.Process[_nProcess].StationFirst  := 26;
      GVL_PROCESS.Process[_nProcess].StationLast   := 37;
      GVL_PROCESS.Process[_nProcess].TargetFirst   := 51;
      GVL_PROCESS.Process[_nProcess].TargetLast    := 51;

      // OUTPUT_R2
      _nProcess                        := OUTPUT_R2;
      GVL_PROCESS.Process[_nProcess].ProcessType   := E_PROCESS_TYPE.PARALLEL_STRICT;
      GVL_PROCESS.Process[_nProcess].StationFirst  := 38;
      GVL_PROCESS.Process[_nProcess].StationLast   := 49;
      GVL_PROCESS.Process[_nProcess].TargetFirst   := 51;
      GVL_PROCESS.Process[_nProcess].TargetLast    := 51;

      // DISTRIBUTOR_1
      _nProcess                        := DISTRIBUTOR_1;
      GVL_PROCESS.Process[_nProcess].ProcessType   := E_PROCESS_TYPE.DISTRIBUTOR;
      GVL_PROCESS.Process[_nProcess].StationFirst  := 50;
      GVL_PROCESS.Process[_nProcess].StationLast   := 50;
      GVL_PROCESS.Process[_nProcess].TargetFirst   := 51;
      GVL_PROCESS.Process[_nProcess].TargetLast    := 51;

      // DISTRIBUTOR_2
      _nProcess                        := DISTRIBUTOR_2;
      GVL_PROCESS.Process[_nProcess].ProcessType   := E_PROCESS_TYPE.DISTRIBUTOR;
      GVL_PROCESS.Process[_nProcess].StationFirst  := 51;
      GVL_PROCESS.Process[_nProcess].StationLast   := 51;
      GVL_PROCESS.Process[_nProcess].TargetFirst   := 52;
      GVL_PROCESS.Process[_nProcess].TargetLast    := 52;
END_METHOD

ACTION StationParameterInit:
//-----------------------------------------------------------------------------
//
//  HAUD 2024.06.12
//
// 
//  - hard coded station parameter
//-----------------------------------------------------------------------------
//-----------------------------------------------------------------------------

//-----------------------------------------------------------------------------------------------------------------------------------------
//  INPUT
    sStationText  := 'INPUT';
//-----------------------------------------------------------------------------------------------------------------------------------------
nStationParameter := 1;
GVL_XTS.StationParameter[nStationParameter].sText                 := sStationText;
GVL_XTS.StationParameter[nStationParameter].rPosWait              :=    988.0;  // absolute modulo position


//-----------------------------------------------------------------------------------------------------------------------------------------
nStationParameter := 2;
GVL_XTS.StationParameter[nStationParameter].sText                 := sStationText;
GVL_XTS.StationParameter[nStationParameter].rPosWait              :=    988.0; // absolute modulo position


//-----------------------------------------------------------------------------------------------------------------------------------------
nStationParameter := 3;
GVL_XTS.StationParameter[nStationParameter].sText                 := sStationText;
GVL_XTS.StationParameter[nStationParameter].rPosWait              :=    988.0; // absolute modulo position


//-----------------------------------------------------------------------------------------------------------------------------------------
nStationParameter := 4;
GVL_XTS.StationParameter[nStationParameter].sText                 := sStationText;
GVL_XTS.StationParameter[nStationParameter].rPosWait              :=   988.0;  // absolute modulo position


//-----------------------------------------------------------------------------------------------------------------------------------------
nStationParameter := 5;
GVL_XTS.StationParameter[nStationParameter].sText                 := sStationText;
GVL_XTS.StationParameter[nStationParameter].rPosWait              :=   988.0;  // absolute modulo position


//-----------------------------------------------------------------------------------------------------------------------------------------
nStationParameter := 6;
GVL_XTS.StationParameter[nStationParameter].sText                 := sStationText;
GVL_XTS.StationParameter[nStationParameter].rPosWait              :=   988.0;  // absolute modulo position


//-----------------------------------------------------------------------------------------------------------------------------------------
nStationParameter := 7;
GVL_XTS.StationParameter[nStationParameter].sText                 := sStationText;
GVL_XTS.StationParameter[nStationParameter].rPosWait              :=   988.0;  // absolute modulo position


//-----------------------------------------------------------------------------------------------------------------------------------------
nStationParameter := 8;
GVL_XTS.StationParameter[nStationParameter].sText                 := sStationText;
GVL_XTS.StationParameter[nStationParameter].rPosWait              :=   988.0;  // absolute modulo position


//-----------------------------------------------------------------------------------------------------------------------------------------
nStationParameter := 9;
GVL_XTS.StationParameter[nStationParameter].sText                 := sStationText;
GVL_XTS.StationParameter[nStationParameter].rPosWait              :=   988.0;  // absolute modulo position


//-----------------------------------------------------------------------------------------------------------------------------------------
nStationParameter := 10;
GVL_XTS.StationParameter[nStationParameter].sText                 := sStationText;
GVL_XTS.StationParameter[nStationParameter].rPosWait              :=   988.0;  // absolute modulo position


//-----------------------------------------------------------------------------------------------------------------------------------------
nStationParameter := 11;
GVL_XTS.StationParameter[nStationParameter].sText                 := sStationText;
GVL_XTS.StationParameter[nStationParameter].rPosWait              :=   988.0;  // absolute modulo position


//-----------------------------------------------------------------------------------------------------------------------------------------
nStationParameter := 12;
GVL_XTS.StationParameter[nStationParameter].sText                 := sStationText;
GVL_XTS.StationParameter[nStationParameter].rPosWait              :=   988.0;  // absolute modulo position


//-----------------------------------------------------------------------------------------------------------------------------------------
//-----------------------------------------------------------------------------------------------------------------------------------------
//  OUTPUT_1
    sStationText  := 'OUTPUT_1';
//-----------------------------------------------------------------------------------------------------------------------------------------
nStationParameter := 13;
GVL_XTS.StationParameter[nStationParameter].sText                 := sStationText;
GVL_XTS.StationParameter[nStationParameter].rPosWait              :=   3582.0;  // absolute modulo position


//-----------------------------------------------------------------------------------------------------------------------------------------
nStationParameter := 14;
GVL_XTS.StationParameter[nStationParameter].sText                 := sStationText;
GVL_XTS.StationParameter[nStationParameter].rPosWait              :=   3582.0;  // absolute modulo position


//-----------------------------------------------------------------------------------------------------------------------------------------
nStationParameter := 15;
GVL_XTS.StationParameter[nStationParameter].sText                 := sStationText;
GVL_XTS.StationParameter[nStationParameter].rPosWait              :=   3582.0;  // absolute modulo position


//-----------------------------------------------------------------------------------------------------------------------------------------
nStationParameter := 16;
GVL_XTS.StationParameter[nStationParameter].sText                 := sStationText;
GVL_XTS.StationParameter[nStationParameter].rPosWait              :=   3582.0;  // absolute modulo position


//-----------------------------------------------------------------------------------------------------------------------------------------
nStationParameter := 17;
GVL_XTS.StationParameter[nStationParameter].sText                 := sStationText;
GVL_XTS.StationParameter[nStationParameter].rPosWait              :=   3582.0;  // absolute modulo position


//-----------------------------------------------------------------------------------------------------------------------------------------
nStationParameter := 18;
GVL_XTS.StationParameter[nStationParameter].sText                 := sStationText;
GVL_XTS.StationParameter[nStationParameter].rPosWait              :=   3582.0;  // absolute modulo position


//-----------------------------------------------------------------------------------------------------------------------------------------
nStationParameter := 19;
GVL_XTS.StationParameter[nStationParameter].sText                 := sStationText;
GVL_XTS.StationParameter[nStationParameter].rPosWait              :=   3582.0;  // absolute modulo position


//-----------------------------------------------------------------------------------------------------------------------------------------
nStationParameter := 20;
GVL_XTS.StationParameter[nStationParameter].sText                 := sStationText;
GVL_XTS.StationParameter[nStationParameter].rPosWait              :=   3582.0;  // absolute modulo position


//-----------------------------------------------------------------------------------------------------------------------------------------
nStationParameter := 21;
GVL_XTS.StationParameter[nStationParameter].sText                 := sStationText;
GVL_XTS.StationParameter[nStationParameter].rPosWait              :=   3582.0;  // absolute modulo position


//-----------------------------------------------------------------------------------------------------------------------------------------
nStationParameter := 22;
GVL_XTS.StationParameter[nStationParameter].sText                 := sStationText;
GVL_XTS.StationParameter[nStationParameter].rPosWait              :=   3582.0;  // absolute modulo position


//-----------------------------------------------------------------------------------------------------------------------------------------
nStationParameter := 23;
GVL_XTS.StationParameter[nStationParameter].sText                 := sStationText;
GVL_XTS.StationParameter[nStationParameter].rPosWait              :=   3582.0;  // absolute modulo position


//-----------------------------------------------------------------------------------------------------------------------------------------
nStationParameter := 24;
GVL_XTS.StationParameter[nStationParameter].sText                 := sStationText;
GVL_XTS.StationParameter[nStationParameter].rPosWait              :=   3582.0;  // absolute modulo position


//-----------------------------------------------------------------------------------------------------------------------------------------
//-----------------------------------------------------------------------------------------------------------------------------------------
//  BUFFER_3
    sStationText  := 'BUFFER_3';
//-----------------------------------------------------------------------------------------------------------------------------------------
nStationParameter := 25;
GVL_XTS.StationParameter[nStationParameter].sText                 := sStationText;
GVL_XTS.StationParameter[nStationParameter].rPosWait              :=   6000.0;  // absolute modulo position


//-----------------------------------------------------------------------------------------------------------------------------------------
//-----------------------------------------------------------------------------------------------------------------------------------------
//  OUTPUT_R1
    sStationText  := 'OUTPUT_R1';
//-----------------------------------------------------------------------------------------------------------------------------------------
nStationParameter := 26;
GVL_XTS.StationParameter[nStationParameter].sText                 := sStationText;
GVL_XTS.StationParameter[nStationParameter].rPosWait              :=   7000.0;  // absolute modulo position


//-----------------------------------------------------------------------------------------------------------------------------------------
nStationParameter := 27;
GVL_XTS.StationParameter[nStationParameter].sText                 := sStationText;
GVL_XTS.StationParameter[nStationParameter].rPosWait              :=   7000.0;  // absolute modulo position


//-----------------------------------------------------------------------------------------------------------------------------------------
nStationParameter := 28;
GVL_XTS.StationParameter[nStationParameter].sText                 := sStationText;
GVL_XTS.StationParameter[nStationParameter].rPosWait              :=   7000.0;  // absolute modulo position


//-----------------------------------------------------------------------------------------------------------------------------------------
nStationParameter := 29;
GVL_XTS.StationParameter[nStationParameter].sText                 := sStationText;
GVL_XTS.StationParameter[nStationParameter].rPosWait              :=   7000.0;  // absolute modulo position


//-----------------------------------------------------------------------------------------------------------------------------------------
nStationParameter := 30;
GVL_XTS.StationParameter[nStationParameter].sText                 := sStationText;
GVL_XTS.StationParameter[nStationParameter].rPosWait              :=   7000.0;  // absolute modulo position


//-----------------------------------------------------------------------------------------------------------------------------------------
nStationParameter := 31;
GVL_XTS.StationParameter[nStationParameter].sText                 := sStationText;
GVL_XTS.StationParameter[nStationParameter].rPosWait              :=   7000.0;  // absolute modulo position


//-----------------------------------------------------------------------------------------------------------------------------------------
nStationParameter := 32;
GVL_XTS.StationParameter[nStationParameter].sText                 := sStationText;
GVL_XTS.StationParameter[nStationParameter].rPosWait              :=   7000.0;  // absolute modulo position


//-----------------------------------------------------------------------------------------------------------------------------------------
nStationParameter := 33;
GVL_XTS.StationParameter[nStationParameter].sText                 := sStationText;
GVL_XTS.StationParameter[nStationParameter].rPosWait              :=   7000.0;  // absolute modulo position


//-----------------------------------------------------------------------------------------------------------------------------------------
nStationParameter := 34;
GVL_XTS.StationParameter[nStationParameter].sText                 := sStationText;
GVL_XTS.StationParameter[nStationParameter].rPosWait              :=   7000.0;  // absolute modulo position


//-----------------------------------------------------------------------------------------------------------------------------------------
nStationParameter := 35;
GVL_XTS.StationParameter[nStationParameter].sText                 := sStationText;
GVL_XTS.StationParameter[nStationParameter].rPosWait              :=   7000.0;  // absolute modulo position


//-----------------------------------------------------------------------------------------------------------------------------------------
nStationParameter := 36;
GVL_XTS.StationParameter[nStationParameter].sText                 := sStationText;
GVL_XTS.StationParameter[nStationParameter].rPosWait              :=   7000.0;  // absolute modulo position


//-----------------------------------------------------------------------------------------------------------------------------------------
nStationParameter := 37;
GVL_XTS.StationParameter[nStationParameter].sText                 := sStationText;
GVL_XTS.StationParameter[nStationParameter].rPosWait              :=   7000.0;  // absolute modulo position


//-----------------------------------------------------------------------------------------------------------------------------------------
//-----------------------------------------------------------------------------------------------------------------------------------------
//  OUTPUT_R2
    sStationText  := 'OUTPUT_R2';
//-----------------------------------------------------------------------------------------------------------------------------------------
nStationParameter := 38;
GVL_XTS.StationParameter[nStationParameter].sText                 := sStationText;
GVL_XTS.StationParameter[nStationParameter].rPosWait              :=   7000.0;  // absolute modulo position


//-----------------------------------------------------------------------------------------------------------------------------------------
nStationParameter := 39;
GVL_XTS.StationParameter[nStationParameter].sText                 := sStationText;
GVL_XTS.StationParameter[nStationParameter].rPosWait              :=   7000.0;  // absolute modulo position


//-----------------------------------------------------------------------------------------------------------------------------------------
nStationParameter := 40;
GVL_XTS.StationParameter[nStationParameter].sText                 := sStationText;
GVL_XTS.StationParameter[nStationParameter].rPosWait              :=   7000.0;  // absolute modulo position


//-----------------------------------------------------------------------------------------------------------------------------------------
nStationParameter := 41;
GVL_XTS.StationParameter[nStationParameter].sText                 := sStationText;
GVL_XTS.StationParameter[nStationParameter].rPosWait              :=   7000.0;  // absolute modulo position


//-----------------------------------------------------------------------------------------------------------------------------------------
nStationParameter := 42;
GVL_XTS.StationParameter[nStationParameter].sText                 := sStationText;
GVL_XTS.StationParameter[nStationParameter].rPosWait              :=   7000.0;  // absolute modulo position


//-----------------------------------------------------------------------------------------------------------------------------------------
nStationParameter := 43;
GVL_XTS.StationParameter[nStationParameter].sText                 := sStationText;
GVL_XTS.StationParameter[nStationParameter].rPosWait              :=   7000.0;  // absolute modulo position


//-----------------------------------------------------------------------------------------------------------------------------------------
nStationParameter := 44;
GVL_XTS.StationParameter[nStationParameter].sText                 := sStationText;
GVL_XTS.StationParameter[nStationParameter].rPosWait              :=   7000.0;  // absolute modulo position


//-----------------------------------------------------------------------------------------------------------------------------------------
nStationParameter := 45;
GVL_XTS.StationParameter[nStationParameter].sText                 := sStationText;
GVL_XTS.StationParameter[nStationParameter].rPosWait              :=   7000.0;  // absolute modulo position


//-----------------------------------------------------------------------------------------------------------------------------------------
nStationParameter := 46;
GVL_XTS.StationParameter[nStationParameter].sText                 := sStationText;
GVL_XTS.StationParameter[nStationParameter].rPosWait              :=   7000.0;  // absolute modulo position


//-----------------------------------------------------------------------------------------------------------------------------------------
nStationParameter := 47;
GVL_XTS.StationParameter[nStationParameter].sText                 := sStationText;
GVL_XTS.StationParameter[nStationParameter].rPosWait              :=   7000.0;  // absolute modulo position


//-----------------------------------------------------------------------------------------------------------------------------------------
nStationParameter := 48;
GVL_XTS.StationParameter[nStationParameter].sText                 := sStationText;
GVL_XTS.StationParameter[nStationParameter].rPosWait              :=   7000.0;  // absolute modulo position


//-----------------------------------------------------------------------------------------------------------------------------------------
nStationParameter := 49;
GVL_XTS.StationParameter[nStationParameter].sText                 := sStationText;
GVL_XTS.StationParameter[nStationParameter].rPosWait              :=   7000.0;  // absolute modulo position



//-----------------------------------------------------------------------------------------------------------------------------------------
//-----------------------------------------------------------------------------------------------------------------------------------------
//  DISTRIBUTOR_1
    sStationText  := 'DISTRIBUTOR_1';
//-----------------------------------------------------------------------------------------------------------------------------------------
nStationParameter := 50;
GVL_XTS.StationParameter[nStationParameter].sText                 := sStationText;
GVL_XTS.StationParameter[nStationParameter].rPosWait              :=  10000.0;  // absolute modulo position


//-----------------------------------------------------------------------------------------------------------------------------------------
//-----------------------------------------------------------------------------------------------------------------------------------------
// DISTRIBUTOR_2
    sStationText  := 'DISTRIBUTOR_2';
//-----------------------------------------------------------------------------------------------------------------------------------------
nStationParameter := 51;
GVL_XTS.StationParameter[nStationParameter].sText                 := sStationText;
GVL_XTS.StationParameter[nStationParameter].rPosWait              :=  11500.0;  // absolute modulo position


//-----------------------------------------------------------------------------------------------------------------------------------------
//-----------------------------------------------------------------------------------------------------------------------------------------
//  BUFFER_4
    sStationText  := 'BUFFER_4';
//-----------------------------------------------------------------------------------------------------------------------------------------
nStationParameter := 52;
GVL_XTS.StationParameter[nStationParameter].sText                 := sStationText;
GVL_XTS.StationParameter[nStationParameter].rPosWait              :=  20000.0;  // absolute modulo position


//-----------------------------------------------------------------------------------------------------------------------------------------
//-----------------------------------------------------------------------------------------------------------------------------------------
//  BUFFER_1
    sStationText  := 'BUFFER_1';
//-----------------------------------------------------------------------------------------------------------------------------------------
nStationParameter := 53;
GVL_XTS.StationParameter[nStationParameter].sText                 := sStationText;
GVL_XTS.StationParameter[nStationParameter].rPosWait              :=    150.0;  // absolute modulo position
END_ACTION

METHOD VisuData
VAR_INPUT
END_VAR

// get enumerations from XPU for visu:
eTransportState                       := f_GetState   (GVL_XTS.XtsTransportState.State);
eTransportResult                      := f_GetProgress(GVL_XTS.XtsTransportState.State);

eXpuState                             := f_GetState   (GVL_XTS.XtsTransportState.XpuState.State);
eXpuResult                            := f_GetProgress(GVL_XTS.XtsTransportState.XpuState.State);

eXpuCheck                             := GVL_XTS.XtsTransportState.XpuState.Check;

// display xpu state and result in visu
// get strings and info
sCaGroupState                         := TO_STRING(GVL_XTS.XtsTransportState.GroupInfo.CaGroupState);

sTransportState                       := TO_STRING(eTransportState);
sTransportCheck                       := TO_STRING(GVL_XTS.XtsTransportState.Check);
sTransportResult                      := TO_STRING(eTransportResult);

sXpuState                             := TO_STRING(eXpuState);
sXpuResult                            := TO_STRING(eXpuResult);
sXpuCheck                             := TO_STRING(eXpuCheck);

sXpuOpMode                            := f_XpuOperationModeToString         (GVL_XTS.XtsTransportState.XpuInfo.OperationMode);
sXpuMoverdetectionMode                := f_MoverIdDetectionModeToString     (GVL_XTS.XtsTransportState.XpuInfo.IdDetectionMode);
sXpuMoverAssignement                  := f_MoverPositionAssignementToString (GVL_XTS.XtsTransportState.XpuInfo.MoverPositionAssignement);

nMoverSelected                        := SEL((nMoverSelected<1), nMoverSelected, 1);
nMoverSelected                        := SEL((nMoverSelected>MAX_MOVER), nMoverSelected, MAX_MOVER);

nStationSelected                      := SEL((nStationSelected<1), nStationSelected, 1);
nStationSelected                      := SEL((nStationSelected>MAX_STATION), nStationSelected, MAX_STATION);

nProcessSelected                      := SEL((nProcessSelected<1), nProcessSelected, 1);
nProcessSelected                      := SEL((nProcessSelected>MAX_PROCESS), nProcessSelected, MAX_PROCESS);

bStationEnable                        := SEL((GVL_XTS.StationCtrl[nStationSelected].eCmd = E_STATION_CTRL.STATION_ENABLE),        FALSE, TRUE);
bStationEnter                         := SEL((GVL_XTS.StationCtrl[nStationSelected].eCmd = E_STATION_CTRL.STATION_MOVER_ENTER),   FALSE, TRUE);
bStationStart                         := SEL((GVL_XTS.StationCtrl[nStationSelected].eCmd = E_STATION_CTRL.STATION_PROCESS_START), FALSE, TRUE);
bStationDone                          := SEL((GVL_XTS.StationCtrl[nStationSelected].eCmd = E_STATION_CTRL.STATION_PROCESS_DONE),  FALSE, TRUE);
bStationOut                           := SEL((GVL_XTS.StationCtrl[nStationSelected].eCmd = E_STATION_CTRL.STATION_MOVER_OUT),     FALSE, TRUE);
bStationGone                          := SEL((GVL_XTS.StationCtrl[nStationSelected].eCmd = E_STATION_CTRL.STATION_MOVER_GONE),    FALSE, TRUE);

sStationState                         := TO_STRING(GVL_XTS.StationState[nStationSelected].eState);
sStationStateMask                     := Tc2_Utilities.BYTE_TO_BINSTR(GVL_XTS.StationState[nStationSelected].nMask, 8);
sStationCtrlMask                      := Tc2_Utilities.BYTE_TO_BINSTR(GVL_XTS.StationCtrl[nStationSelected].nMask, 8);

sProcessEnableMask                    := Tc2_Utilities.WORD_TO_BINSTR(GVL_PROCESS.Process[nProcessSelected].EnableProcess, 16);
END_METHOD

END_PROGRAM

// ---- XTS_TRANSPORT/_types/f_GetProgress.TcPOU
// global function to extract e_progress from combined value
FUNCTION f_GetProgress : uint
VAR_INPUT
  state     : UINT;
END_VAR
VAR
  nP        : uint;
END_VAR


nP := state / E_PROGRESS.PROGRESS_INIT;

f_GetProgress := nP * E_PROGRESS.PROGRESS_INIT;

END_FUNCTION

// ---- PROCESS/fb_Process.TcPOU
//---------------------------------------------------------------------------------------------------------------
//
//  HAUD 2023.03.27
//
//  TR08
//  - XTS_TRANSPORT_LAYER
//
//  fb_Process
//  - grouping of xts stations to sync start process
//  - nFirst to nLast xts stations are checked for starting process simultaneously
//  - basic preparation of station target index in PrepareTarget()
//  - handshake with station control for mover transport through station
//
//---------------------------------------------------------------------------------------------------------------
// This SOFTWARE is provided as an Exemple by THE PROVIDER "as is" and "with all faults." THE PROVIDER makes no 
// representations or warranties of any kind concerning the safety, suitability, lack of viruses, inaccuracies, 
// typographical errors, or other harmful components of this SOFTWARE. There are inherent dangers in the use of 
// any software, and you are solely responsible for determining whether this SOFTWARE is compatible with your 
// equipment and other software installed on your equipment. You are also solely responsible for the protection 
// of your equipment and backup of your data, and THE PROVIDER will not be liable for any damages you may suffer 
// in connection with using, modifying, or distributing this SOFTWARE.
//---------------------------------------------------------------------------------------------------------------
FUNCTION_BLOCK fb_Process IMPLEMENTS I_ExternControl_Process
VAR
  _eType                      : E_PROCESS_TYPE;   // types of process: SINGLE, PARALLEL, SERIAL, DISTRIBUTOR
  _sCheck                     : STRING;

  _eProcessCmd                : E_STATION_CTRL;   // control from property
  _eProcessState              : E_STATION_STATE;  // state   to   property

  {attribute 'displaymode':='bin'}
  _wEnableProcess             : WORD; // control sets bits to switch on stations
  _bEnabledStation            : POINTER TO ARRAY[1..XTS_Parameter.MAX_STATION]  OF BOOL; // information about all enabled xts stations

  // xts stations
  _stCtrl                     : POINTER TO ARRAY[1..XTS_Parameter.MAX_STATION]  OF ST_STATION_CTRL;
  _stState                    : POINTER TO ARRAY[1..XTS_Parameter.MAX_STATION]  OF ST_STATION_STATE;

  // who is included in process
  // _nFirst to _nLast MUST be in closed consecutive order
  _nStation,
  _nStationCount,
  _nFirstStation,
  _nLastStation               : UINT;

  // work vars for writing onto _stCtrl[nStation].nTargetStation
  _nTarget,
  _nFirstTarget,
  _nLastTarget                : UINT;   // for parallel process xts stations and the last xts station in serial process

  _nSerialTarget              : ARRAY[1..XTS_Parameter.MAX_STATION]  OF UINT; // serial targets within process

  _nPreparedTarget            : ARRAY[1..XTS_Parameter.MAX_MOVER]  OF UINT;   // targets for parallel and single process

  // bitmasks for station states in CycleStation()
  {attribute 'displaymode':='bin'}
  _wEnable                    : WORD;   // commanded enable of xts station
  {attribute 'displaymode':='bin'}
  _wEnter                     : WORD;   // mover asking for entry into xts station
  {attribute 'displaymode':='bin'}
  _wStart                     : WORD;   // xts station asking for process handshake
  {attribute 'displaymode':='bin'}
  _wLeave                     : WORD;   // xts station wants to send out mover
  {attribute 'displaymode':='bin'}
  _wQueue                     : WORD;   // mover was entered into xts station list
  {attribute 'displaymode':='bin'}
  _wMoverInStation            : WORD;   // mover entry was granted, mover is now in station
  {attribute 'displaymode':='bin'}
  _wError                     : WORD;   // minor error, must be fixed by _stCtrl[nStation]
  {attribute 'displaymode':='bin'}
  _wErrorFatal                : WORD;   // fatal error, must be fixed by debugging
  {attribute 'displaymode':='bin'}
  _wTargetId                  : WORD;   // nTargetStation > 0 in _stDtrl[nStation].nTargetStation

  {attribute 'displaymode':='bin'}
  _TargetMask                 : DWORD;   // bit positions correspond to index of xts station
 
  _bNext                      : BOOL;

  _nProcessPerMinute          : uint; // sum of all xts stations output per minute in process
  _rtrigProcess               : ARRAY[1..XTS_Parameter.MAX_STATION] OF Tc2_Standard.R_TRIG;
  _tonPartsPerMinute          : Tc2_Standard.TON;

  _nMoverPerMinute            : POINTER TO ARRAY[1..XTS_Parameter.MAX_STATION]  OF UINT;
  _nMoverCount,
  _nMoverCountOld             : ARRAY[1..XTS_Parameter.MAX_STATION]  OF UINT;

  _eDistributorTarget         : E_PROGRESS;

END_VAR

METHOD private Check : BOOL

IF (_nFirstStation < 1) OR
   (_nFirstStation > MAX_STATION)
THEN
  _sCheck                     := '_nFirstStation out of bounds';
  RETURN;
END_IF

IF (_nLastStation < 1) OR
   (_nLastStation > MAX_STATION)
THEN
  _sCheck                     := '_nLastStation out of bounds';
  RETURN;
END_IF

IF (_nFirstTarget < 1) OR
   (_nFirstTarget > MAX_STATION)
THEN
  _sCheck                     := '_nFirstTarget out of bounds';
  RETURN;
END_IF

IF (_nLastTarget < 1) OR
   (_nLastTarget > MAX_STATION)
THEN
  _sCheck                     := '_nLastTarget out of bounds';
  RETURN;
END_IF

IF NOT (_stCtrl  <> 0)
THEN
  _sCheck                     := '_stCtrl: missing pointer';
  RETURN;
END_IF

IF NOT (_stState <> 0)
THEN
  _sCheck                     := '_stState: missing pointer';
  RETURN;
END_IF

IF NOT (_bEnabledStation  <> 0)
THEN
  _sCheck                     := '_bEnableStation: missing pointer';
  RETURN;
END_IF

IF not (_nMoverPerMinute <> 0)
THEN
  _sCheck                     := '_nMoverPerMinute: missing pointer';
  RETURN;
END_IF

_nStationCount                := _nLastStation - _nFirstStation + 1;

IF (_nStationCount < 1) OR
   (_nStationCount > (SIZEOF(WORD)*8))
THEN
  _sCheck                     := '_nStationCount out of bounds';
  RETURN;
END_IF


_sCheck                       := TO_STRING(E_PROGRESS.PROGRESS_DONE);
Check                         := TRUE;
END_METHOD

METHOD Cycle
VAR_INST
  _nStn     : uint;
END_VAR
IF NOT Check() THEN RETURN; END_IF


//-----------------------------------------------------------------------------
// collect state information from xts stations
// state information is collected in Masks (WORD), 
// every bit represents one XTS station in process
//-----------------------------------------------------------------------------
//  _wEnable                        : enable cmd was given to xts station
//  _wEnter                         : a mover is requesting entry
//  _wStart                         : mover has arrived and xts station is ready
//  _wLeave                         : xts station wants to send mover out
//  _wQueue                         : somebody's waiting
//  _wMoverInStation                : mover is in station
//  _wError                         : error state for handshake
//  _wErrorFatal                    : error state for severe problems (debugging required)
//  _wTargetId                      : Ctrl.nTargetStation > 0
//  _wMoverInQueueSerial            : SERIAL process: bits to check whether a mover is waiting to be processed
//
CycleStation();                     // get state information from all XtsStations in process
//-----------------------------------------------------------------------------
//-----------------------------------------------------------------------------
//  E_STATION_CTRL.STATION_INIT: hard reset of process and XtsStations
//-----------------------------------------------------------------------------
CASE _eProcessCmd                   // check input property
OF
  E_STATION_CTRL.STATION_INIT:      // commanded init from ctrl
    CASE _eType
    OF
      E_PROCESS_TYPE.SERIAL:
        InitSerialTargets();
    END_CASE
    Init();                         RETURN; // rest you will, return you must
END_CASE
//-----------------------------------------------------------------------------
// E_STATION_STATE.STATION_INIT: pass through here and switch off XtsStations
//-----------------------------------------------------------------------------
CASE _eProcessState                 // check output property
OF
  E_STATION_STATE.STATION_INIT:     // xts station empty, disabled by default
    _eProcessState                  := E_STATION_STATE.STATION_DISABLE;
    FOR _nStn := _nLastStation TO _nFirstStation BY(-1) 
    DO
      _stCtrl^[_nStn].eCmd          := E_STATION_CTRL.STATION_DISABLE;
    END_FOR

END_CASE
//-----------------------------------------------------------------------------
//  E_STATION_STATE.STATION_DISABLE: wait for enable from flow control
//-----------------------------------------------------------------------------
CASE _eProcessState                 // check output property
OF
  E_STATION_STATE.STATION_DISABLE:  // check for enable command
    IF (_eProcessCmd = E_STATION_CTRL.STATION_ENABLE)
    THEN
      _eProcessState                := E_STATION_STATE.STATION_ENABLE;

      FOR _nStn := _nLastStation TO _nFirstStation BY(-1) 
      DO
          _stCtrl^[_nStn].eCmd      := E_STATION_CTRL.STATION_ENABLE;
      END_FOR
    END_IF
END_CASE
//-----------------------------------------------------------------------------
//  E_STATION_STATE.STATION_ENABLE: check Cmd and wait for XtsStations to be enabled
//-----------------------------------------------------------------------------
CASE _eProcessState
OF
  E_STATION_STATE.STATION_ENABLE:
    CASE _eProcessCmd
    OF
      E_STATION_CTRL.STATION_DISABLE:
        _eProcessState              := E_STATION_STATE.STATION_INIT;

      E_STATION_CTRL.STATION_ENABLE:
        IF (_wEnable = _wEnableProcess)
        THEN
          InitSerialTargets();
          _eProcessState            := E_STATION_STATE.STATION_DETECT_MOVER;
        END_IF
    END_CASE
END_CASE
//-----------------------------------------------------------------------------
// E_STATION_STATE.STATION_DETECT_MOVER: wait for any XtsStation to 
//                                       have a mover ready to enter
//-----------------------------------------------------------------------------
CASE _eProcessState
OF
  E_STATION_STATE.STATION_DETECT_MOVER:
    CASE _eProcessCmd
    OF
      E_STATION_CTRL.STATION_DISABLE:
        _eProcessState              := E_STATION_STATE.STATION_INIT;

      E_STATION_CTRL.STATION_ENABLE:
        IF (_wEnter > 0)            // at least one mover is asking for entry
        THEN
          _eDistributorTarget       := E_PROGRESS.PROGRESS_INVALID;

                                    // switch process state in order to tell process control
          _eProcessState            := E_STATION_STATE.STATION_MOVER_ENTER;
        END_IF
    END_CASE
END_CASE
//-----------------------------------------------------------------------------
//  E_STATION_STATE.STATION_MOVER_ENTER: check if infeed conditions are met, 
//                                       depending on type of process
//                                       Cmd from input (flow control)
//-----------------------------------------------------------------------------
CASE _eProcessState
OF
  E_STATION_STATE.STATION_MOVER_ENTER:
    CASE _eProcessCmd               // check input property
    OF
      E_STATION_CTRL.STATION_DISABLE:
        _eProcessState              := E_STATION_STATE.STATION_INIT;

      E_STATION_CTRL.STATION_MOVER_ENTER:
        FOR _nStn := _nLastStation TO _nFirstStation BY(-1) 
        DO
          CASE _stState^[_nStn].eState
          OF
          E_STATION_STATE.STATION_MOVER_ENTER,
          E_STATION_STATE.STATION_MOVER_IN_TARGET,
          E_STATION_STATE.STATION_PROCESS_START:
            IF GetBitWord(_wEnter, (_nStn - _nFirstStation))
            THEN
              _stCtrl^[_nStn].eCmd  := E_STATION_CTRL.STATION_MOVER_ENTER;
            END_IF
          ELSE
            IF _bEnabledStation^[_nStn]
            THEN
              _stCtrl^[_nStn].eCmd  := E_STATION_CTRL.STATION_ENABLE;
            END_IF
          END_CASE
        END_FOR

        CASE _eType
        OF
          E_PROCESS_TYPE.PARALLEL_STRICT:
            IF (_wStart = _wEnable) // all who are enabled must have mover, in order to continue
            THEN
              _eProcessState        := E_STATION_STATE.STATION_PROCESS_START;
            END_IF

          E_PROCESS_TYPE.PARALLEL: 
            IF (_wStart = _wEnter)
            THEN
              _eProcessState        := E_STATION_STATE.STATION_PROCESS_START;
            END_IF

          E_PROCESS_TYPE.SERIAL:    // all who have work to do must have mover, in order to continue
            IF (_wMoverInStation > 0)
            THEN
              IF (_wStart = _wMoverInStation)
              THEN
                _eProcessState      := E_STATION_STATE.STATION_PROCESS_START;
              END_IF
            END_IF
        ELSE
          _eProcessState            := E_STATION_STATE.STATION_PROCESS_START;
        END_CASE

      E_STATION_CTRL.STATION_MOVER_SEND:  // flow control decided to skip process
        FOR _nStn := _nLastStation TO _nFirstStation BY(-1) 
        DO
          IF _bEnabledStation^[_nStn] AND 
             GetBitWord(_wQueue, (_nStn-_nFirstStation))
          THEN
            IF (_TargetMask > 0)
            THEN
              // station is enabled AND has a mover in Queue to send
              _stCtrl^[_nStn].eCmd    := E_STATION_CTRL.STATION_MOVER_SEND;
            END_IF
          END_IF
        END_FOR
        IF (_wLeave > 0)            // wait for XtsStation to switch to outfeed
        THEN
          IF (_TargetMask > 0)
          THEN
            _eDistributorTarget       := DistributorTarget(_TargetMask);         // prepare target for mover
            IF (_eDistributorTarget = E_PROGRESS.PROGRESS_DONE)
            THEN
              _wStart                 := _wLeave;
              _eProcessState          := E_STATION_STATE.STATION_CHECK;
            END_IF
          END_IF
        END_IF 
    END_CASE
END_CASE
//-----------------------------------------------------------------------------
// synced process handshake on all stations in process
//-----------------------------------------------------------------------------
CASE _eProcessState                 // check output property
OF
  E_STATION_STATE.STATION_PROCESS_START:
    CASE _eType                     // decision for synced start varies for e_process_type
    OF
      E_PROCESS_TYPE.SERIAL:        // serial process must have had a mover waiting, which is now processed
      CASE _eProcessCmd             // check command input property
      OF
        E_STATION_CTRL.STATION_PROCESS_START,
        E_STATION_CTRL.STATION_PROCESS_DONE:
            IF (_wStart = _wMoverInStation)
            THEN
              _eProcessState          := E_STATION_STATE.STATION_PROCESS_DONE;
              FOR _nStn := _nLastStation TO _nFirstStation BY(-1) 
              DO
                // check for correct state on XtsStation
                CASE _stState^[_nStn].eState
                OF
                E_STATION_STATE.STATION_PROCESS_START:
                  _stCtrl^[_nStn].eCmd  := _eProcessCmd;
                END_CASE
              END_FOR
            END_IF
      END_CASE
    ELSE
      CASE _eProcessCmd             // check command input property
      OF
        E_STATION_CTRL.STATION_PROCESS_START,
        E_STATION_CTRL.STATION_PROCESS_DONE:
          IF (_wStart = _wEnter)
          THEN
            _eProcessState          := E_STATION_STATE.STATION_PROCESS_DONE;
            FOR _nStn := _nLastStation TO _nFirstStation BY(-1) 
            DO
              // check for correct state on XtsStation
              CASE _stState^[_nStn].eState
              OF
              E_STATION_STATE.STATION_PROCESS_START:
                _stCtrl^[_nStn].eCmd  := _eProcessCmd;
              END_CASE
            END_FOR
          END_IF
      END_CASE
    END_CASE
END_CASE
//-----------------------------------------------------------------------------
// synced process handshake on all stations in process
//-----------------------------------------------------------------------------
CASE _eProcessState                 // check output property
OF
  E_STATION_STATE.STATION_PROCESS_DONE:
    CASE _eProcessCmd               // check command input property
    OF
      E_STATION_CTRL.STATION_PROCESS_DONE: 
        FOR _nStn := _nLastStation TO _nFirstStation BY(-1) 
        DO
          _stCtrl^[_nStn].eCmd      := E_STATION_CTRL.STATION_PROCESS_DONE;
        END_FOR
        IF (_wLeave > 0)            // _wLeave tells us that xts station has mover to send
        THEN
          CASE _eType
          OF
            E_PROCESS_TYPE.SERIAL:
              _eProcessState        := E_STATION_STATE.STATION_CHECK;
              IF (_stState^[_nLastStation].nMoverId > 0)
              THEN
                PrepareLastSerialTarget();     // target for last xts station in serial process
              END_IF
    
              FOR _nStn := (_nLastStation - 1) TO _nFirstStation BY(-1) 
              DO
                _stCtrl^[_nStn].nTargetStation    := TO_USINT(_nSerialTarget[_nStn]);
              END_FOR
          ELSE
              IF (_TargetMask > 0)
              THEN
                ParallelTargets(_TargetMask);
                _eProcessState      := E_STATION_STATE.STATION_CHECK;
              END_IF
          END_CASE
        END_IF
    END_CASE
END_CASE
//-----------------------------------------------------------------------------
//-----------------------------------------------------------------------------
CASE _eProcessState
OF
  E_STATION_STATE.STATION_CHECK:    // TODO: implement procedure for target plausibility
    IF (_wTargetId > 0)             // simple check any target before switching to outfeed
    THEN
       _eProcessState               := E_STATION_STATE.STATION_MOVER_OUT;
    ELSE                            // in case of invalid target, wait here for retry
      CASE _eType                   // retry varies for e_process_type
      OF
        E_PROCESS_TYPE.DISTRIBUTOR:
          IF (_eProcessCmd = E_STATION_CTRL.STATION_ENABLE)
          THEN
            // only distributor can land here directly; retry mover infeed
            _eProcessState          := E_STATION_STATE.STATION_MOVER_ENTER;
          END_IF
      ELSE
          IF (_eProcessCmd = E_STATION_CTRL.STATION_PROCESS_START)
          THEN
            // all other e_process_type must go back to process handshake
            _eProcessState          := E_STATION_STATE.STATION_PROCESS_DONE;
          END_IF
      END_CASE
    END_IF
END_CASE
//-----------------------------------------------------------------------------
//-----------------------------------------------------------------------------
CASE _eProcessState
OF
  E_STATION_STATE.STATION_MOVER_OUT:
    IF (_wLeave = 0)                // all movers are gone
    THEN
      _eProcessState                := E_STATION_STATE.STATION_MOVER_GONE;

    ELSIF (_wLeave = _wStart)       // wait for everybody to be ready for send out
    THEN
      IF (_eProcessCmd = E_STATION_CTRL.STATION_MOVER_OUT)
      THEN
        FOR _nStn := _nLastStation TO _nFirstStation BY(-1) 
        DO
          CASE _stState^[_nStn].eState  // double check valid xts station state
          OF
            E_STATION_STATE.STATION_MOVER_OUT:
              IF (_stCtrl^[_nStn].nTargetStation > 0) // double check ticket on ctrl struct
              THEN
                _stCtrl^[_nStn].eCmd  := E_STATION_CTRL.STATION_MOVER_OUT;
              END_IF
          END_CASE
        END_FOR
      END_IF
    END_IF
END_CASE
//-----------------------------------------------------------------------------
//-----------------------------------------------------------------------------
CASE _eProcessState
OF
  E_STATION_STATE.STATION_MOVER_GONE:   // station is empty, quit mover gone and go back to the beginning
    FOR _nStn := _nLastStation TO _nFirstStation BY(-1) 
    DO
      _stCtrl^[_nStn].eCmd      := E_STATION_CTRL.STATION_MOVER_GONE;
    END_FOR
    _eProcessState              := E_STATION_STATE.STATION_INIT;
END_CASE
END_METHOD

METHOD PRIVATE CycleStation
VAR
  _k                  : UINT;
END_VAR
IF NOT Check() THEN RETURN; END_IF

_wError                                   :=
_wErrorFatal                              := 0;

FOR _nStation := _nLastStation TO _nFirstStation BY(-1) 
DO
  // copy bit for enable station from input word to global array in GVL_PROCESS,
  //  - other processes read enabled state on mover out (PrepareTarget)
  _bEnabledStation^[_nStation]            := GetBitWord(_wEnableProcess, (_nStation-_nFirstStation));

  IF (_stCtrl^[_nStation].nTargetStation > 0)
  THEN
    _wTargetId                            := SetBitWord(_wTargetId,  (_nStation-_nFirstStation));
  ELSE
    _wTargetId                            := DelBitWord(_wTargetId,  (_nStation-_nFirstStation));
  END_IF

  IF (_stState^[_nStation].nMoverId > 0)
  THEN
    _wMoverInStation                      := SetBitWord(_wMoverInStation,  (_nStation-_nFirstStation));
  ELSE
    _wMoverInStation                      := DelBitWord(_wMoverInStation,  (_nStation-_nFirstStation));
  END_IF

  IF (_stState^[_nStation].nQueue > 0)
  THEN
    _wQueue                               := SetBitWord(_wQueue,  (_nStation-_nFirstStation));
  ELSE
    _wQueue                               := DelBitWord(_wQueue,  (_nStation-_nFirstStation));
  END_IF

  CASE _stCtrl^[_nStation].eCmd
  OF
    E_STATION_CTRL.STATION_INIT:
      _stCtrl^[_nStation].nTargetStation  := 0;
      _wEnable                            := DelBitWord(_wEnable, (_nStation-_nFirstStation));
      _wEnter                             := DelBitWord(_wEnter,  (_nStation-_nFirstStation));
      _wStart                             := DelBitWord(_wStart,  (_nStation-_nFirstStation));
      _wLeave                             := DelBitWord(_wLeave,  (_nStation-_nFirstStation));

    E_STATION_CTRL.STATION_ENABLE:
      _wEnable                            := SetBitWord(_wEnable, (_nStation-_nFirstStation));
  END_CASE

  CASE _stState^[_nStation].eState
  OF
    E_STATION_STATE.STATION_DISABLE:
      _wEnter                             := DelBitWord(_wEnter,  (_nStation-_nFirstStation));

    E_STATION_STATE.STATION_MOVER_ENTER,
    E_STATION_STATE.STATION_MOVER_IN_TARGET:
      _wEnter                             := SetBitWord(_wEnter,  (_nStation-_nFirstStation));
  
    E_STATION_STATE.STATION_PROCESS_START,
    E_STATION_STATE.STATION_PROCESS_DONE:
      _wStart                             := SetBitWord(_wStart,  (_nStation-_nFirstStation));
  
    E_STATION_STATE.STATION_MOVER_OUT:
      _wLeave                             := SetBitWord(_wLeave,  (_nStation-_nFirstStation));


    E_STATION_STATE.STATION_MOVER_GONE:
      _stCtrl^[_nStation].nTargetStation  := 0;
      _wStart                             := DelBitWord(_wStart,  (_nStation-_nFirstStation));
      _wLeave                             := DelBitWord(_wLeave,  (_nStation-_nFirstStation));
      _wEnable                            := DelBitWord(_wEnable, (_nStation-_nFirstStation));
      _wEnter                             := DelBitWord(_wEnter,  (_nStation-_nFirstStation));


    E_STATION_STATE.STATION_ERROR_LIST_STATION_ID_WRONG,  // wrong station ID in mover ticket (nTargetId written by preceeding station/process)
    E_STATION_STATE.STATION_ERROR_OUTFEED_TARGET_INVALID, // write correct target on station Ctrl.nTargetStation
    E_STATION_STATE.STATION_ERROR_INFEED_ERROR,           // clear mover error via Ctrl/State interface and retry on XTS station directly
    E_STATION_STATE.STATION_ERROR_OUTFEED_ERROR:          // clear mover error via Ctrl/State interface and retry on XTS station directly
      _wError                             := SetBitWord(_wError,      (_nStation-_nFirstStation));

    E_STATION_STATE.STATION_ERROR_FATAL:
      _wErrorFatal                        := SetBitWord(_wErrorFatal, (_nStation-_nFirstStation));

  END_CASE
END_FOR


_nProcessPerMinute          := 0;
// get mover counter
FOR _k := _nLastStation TO _nFirstStation BY(-1) 
DO
  _rtrigProcess[_k](
                  CLK       := (_stCtrl^[_k].eCmd = E_STATION_CTRL.STATION_MOVER_OUT));

  IF _rtrigProcess[_k].Q
  THEN
    _nMoverCount[_k]        := _nMoverCount[_k] + 1;
  END_IF
  
  IF _tonPartsperMinute.Q
  THEN
    _nMoverPerMinute^[_k]   := _nMoverCount[_k] - _nMoverCountOld[_k];
    _nMoverCountOld  [_k]   := _nMoverCount[_k];
  END_IF
  _nProcessPerMinute        := _nProcessPerMinute + _nMoverPerMinute^[_k]; 
END_FOR

IF _tonPartsperMinute.q
THEN
  _tonPartsperMinute(
                  IN        :=FALSE);
END_IF

_tonPartsperMinute(
                  IN        := TRUE, 
                  PT        := T#60S);
END_METHOD

METHOD PUBLIC DelBitWord : WORD
VAR_INPUT
  inVal   : WORD;
  bitNo   : DINT;
END_VAR
VAR
  wConst : WORD := 1;
END_VAR
IF ( inVal AND SHL( wConst,bitNo MOD 16 ) ) > 0 THEN
  DelBitWord := inVal XOR (SHL( wConst,bitNo MOD 16 ));
ELSE
  DelBitWord := inVal;
END_IF
END_METHOD

METHOD DistributorTarget : e_progress
VAR_INPUT
  wTarget         : DWORD; // bits for target stations to be used
END_VAR
VAR_INST
  _eResult        : E_PROGRESS;
  {attribute 'displaymode':='bin'}
  _wtg            : DWORD;
END_VAR
IF NOT Check() THEN RETURN; END_IF
_wtg := wTarget;

// check if target station is enabled
IF GetBitDWord(wTarget, (_nTarget))
THEN
  _nPreparedTarget[_stState^[_nFirstStation].nMoverId]  := _nLastTarget - _nTarget;
  _stCtrl^[_nFirstStation].nTargetStation               := TO_USINT(_nLastTarget - _nTarget);
  _eResult                                              := E_PROGRESS.PROGRESS_DONE;
ELSE
  _eResult                                              := e_progress.PROGRESS_BUSY;
END_IF

_nTarget                      := _nTarget + 1;
IF (_nLastTarget - _nTarget < _nFirstTarget)
THEN
  _nTarget                    := 0;
END_IF

DistributorTarget                                       := _eResult;
END_METHOD

PROPERTY EnabledStation : POINTER TO ARRAY[1..XTS_Parameter.MAX_STATION]  OF bool;
SET
_bEnabledStation := EnabledStation;
END_SET
END_PROPERTY

PROPERTY EnableProcess : word
GET
EnableProcess := _wEnableProcess;
END_GET
SET
_wEnableProcess := EnableProcess;
END_SET
END_PROPERTY

METHOD PUBLIC GetBitDWord : BOOL
VAR_INPUT
  inVal   : DWORD;
  bitNo   : DINT;
END_VAR
VAR
  wConst : DWORD := 1;
END_VAR
IF ( inVal AND SHL( wConst,DINT_TO_SINT(bitNo) MOD 32 ) ) > 0
THEN
  GetBitDWord := TRUE;
ELSE
  GetBitDWord := FALSE;
END_IF
END_METHOD

METHOD PUBLIC GetBitWord : BOOL
VAR_INPUT
  inVal   : WORD;
  bitNo   : DINT;
END_VAR
VAR
  wConst : WORD := 1;
END_VAR
IF ( inVal AND SHL( wConst,DINT_TO_SINT(bitNo) MOD 16 ) ) > 0
THEN
  GetBitWord := TRUE;
ELSE
  GetBitWord := FALSE;
END_IF
END_METHOD

METHOD PUBLIC Init : BOOL
VAR
  _nStn     : UINT;
END_VAR
IF NOT (_nLastStation   > 0) OR
   NOT (_nFirstStation  > 0) OR
   NOT (_nLastStation   < MAX_STATION+1) OR
   NOT (_nFirstStation  < MAX_STATION+1)
THEN
  Init := FALSE;
  _eProcessState                := E_STATION_STATE.STATION_NO_INIT;
ELSE
  _eProcessState                := E_STATION_STATE.STATION_NO_INIT;

  FOR _nStn := _nLastStation TO _nFirstStation BY(-1) 
  DO
    _stCtrl^[_nStn].eCmd        := E_STATION_CTRL.STATION_INIT;
    _stCtrl^[_nStn].nMask       := 0;

    IF NOT (_stState^[_nStn].eState = E_STATION_STATE.STATION_INIT)
    THEN
      Init := FALSE;
      RETURN;
    END_IF  
  END_FOR

  memset(ADR(_nMoverCount),       0, SIZEOF(_nMoverCount));
  memset(ADR(_nMoverCountOld),    0, SIZEOF(_nMoverCountOld));
  _nTarget                      := 0;

  _eProcessState                := E_STATION_STATE.STATION_INIT;

  Init := TRUE;
END_IF
END_METHOD

METHOD PRIVATE InitSerialTargets
VAR
  _k    : uint;
END_VAR

IF NOT (_nStationCount > 1)
THEN
  RETURN;
END_IF

// serial process must always have at least two xts stations to work with
FOR _nStation := _nLastStation TO _nFirstStation+1 BY(-1) 
DO
  IF (_bEnabledStation^[_nStation])
  THEN
    _nSerialTarget[_nStation-1] := _nStation;
  END_IF
END_FOR
END_METHOD

PROPERTY MoverCountInQueue : uint
GET
VAR
  _nTmp   : UINT;
  _nCount : uint;
END_VAR
IF NOT (_nStationCount > 0)
THEN
  MoverCountInQueue := 0;
  RETURN;
END_IF

FOR _nTmp := _nLastStation TO _nFirstStation BY(-1)
DO
  _nCount := _nCount + _stState^[_nTmp].nQueue;
END_FOR

MoverCountInQueue := _nCount;
END_GET
END_PROPERTY

PROPERTY MoverInQueue : Bool
GET
MoverInQueue  := SEL((_wQueue > 0), FALSE, TRUE);
END_GET
END_PROPERTY

PROPERTY MoverPerMinute : pointer to ARRAY[1..XTS_Parameter.MAX_STATION]  OF UINT
SET
_nMoverPerMinute  := MoverPerMinute;
END_SET
END_PROPERTY

METHOD PRIVATE ParallelTargets : E_PROGRESS
VAR_INPUT
  wTarget         : DWORD; // bits for target stations to be used
END_VAR
VAR_INST
  {attribute 'displaymode':='bin'}
  _wtg            : DWORD;
  _nt,
  _idxStation     : UINT;
END_VAR
IF NOT Check() THEN RETURN; END_IF
_wtg := wTarget;


FOR _idxStation := _nLastStation TO _nFirstStation BY(-1) 
DO
  _nt                           := _nLastTarget - _nTarget;

  // check if target station is enabled
  IF GetBitDWord(wTarget, (_nTarget))
  THEN
    IF (_stState^[_idxStation].nMoverId <> 0)
    THEN
      _nPreparedTarget[_stState^[_idxStation].nMoverId]  := _nt;
      _stCtrl^[_idxStation].nTargetStation               := TO_USINT(_nt);
    END_IF
  END_IF

  _nTarget                      := _nTarget + 1;
  IF (_nLastTarget - _nTarget < _nFirstTarget)
  THEN
    _nTarget                    := 0;
  END_IF
END_FOR
END_METHOD

METHOD PRIVATE PrepareLastSerialTarget
VAR
  _nt   : uint;
END_VAR

_nt                           := _nLastTarget - _nTarget;
_nTarget                      := _nTarget + 1;

// check if target station is enabled
IF (_bEnabledStation^[_nt])
THEN
  _nPreparedTarget[_stState^[_nLastStation].nMoverId]  := _nt;
  _stCtrl^[_nLastStation].nTargetStation               := TO_USINT(_nt);
END_IF

IF (_nLastTarget - _nTarget < _nFirstTarget)
THEN
  _nTarget                    := 0;
END_IF
END_METHOD

PROPERTY ProcessCmd : E_STATION_CTRL
SET
_eProcessCmd := ProcessCmd;
END_SET
END_PROPERTY

PROPERTY ProcessPerMinute : uint
GET
ProcessPerMinute := _nProcessPerMinute;
END_GET
END_PROPERTY

PROPERTY ProcessState : E_STATION_STATE
GET
ProcessState := _eProcessState;
END_GET
END_PROPERTY

PROPERTY ProcessType : e_process_type
GET
ProcessType := _eType;
END_GET
SET
_eType := ProcessType;
END_SET
END_PROPERTY

METHOD PUBLIC SetBitDWord : DWORD
VAR_INPUT
  inVal   : DWORD;
  bitNo   : DINT;
END_VAR
VAR
  wConst  : DWORD := 1;
END_VAR
SetBitDWord := inVal OR SHL( wConst,bitNo MOD 32 );
END_METHOD

METHOD PUBLIC SetBitWord : WORD
VAR_INPUT
  inVal   : WORD;
  bitNo   : DINT;
END_VAR
VAR
  wConst  : WORD := 1;
END_VAR
SetBitWord := inVal OR SHL( wConst,bitNo MOD 16 );
END_METHOD

PROPERTY StationCount : uint
GET
StationCount := _nStationCount;
END_GET
END_PROPERTY

PROPERTY StationCtrl : pointer to ARRAY[1..XTS_Parameter.MAX_STATION]  OF ST_STATION_CTRL;
SET
_stCtrl := StationCtrl;
END_SET
END_PROPERTY

PROPERTY StationFirst : uint
GET
StationFirst := _nFirstStation;
END_GET
SET
_nFirstStation := StationFirst;
END_SET
END_PROPERTY

PROPERTY StationLast : uint
GET
StationLast := _nLastStation;
END_GET
SET
_nLastStation := StationLast;
END_SET
END_PROPERTY

PROPERTY StationState : POINTER TO ARRAY[1..XTS_Parameter.MAX_STATION]  OF ST_STATION_STATE
SET
_stState := StationState;
END_SET
END_PROPERTY

PROPERTY TargetFirst : uint
GET
TargetFirst := _nFirstTarget;
END_GET
SET
_nFirstTarget := TargetFirst;
END_SET
END_PROPERTY

PROPERTY TargetLast : uint
GET
TargetLast := _nLastTarget;
END_GET
SET
_nLastTarget := TargetLast;
END_SET
END_PROPERTY

PROPERTY TargetMask : dword
GET
TargetMask := _TargetMask;
END_GET
SET
_TargetMask := TargetMask;
END_SET
END_PROPERTY

END_FUNCTION_BLOCK

// ---- PROCESS/proc/fb_Worker.TcPOU
FUNCTION_BLOCK fb_Worker
VAR
  _nProcess         : UINT;

  _ItfProcess       : REFERENCE TO ARRAY[1..MAX_PROCESS] OF I_ExternControl_Process;

  _tonProcess       : Tc2_Standard.TON;
  _tProcess         : TIME;

  _nMoverPerMinute  : UINT;

  _wTargetMask      : DWORD;
  _nQueue           : ARRAY[1..MAX_PROCESS] OF UINT;

END_VAR

METHOD AUTO : E_PROGRESS
VAR_INPUT
  Active            : BOOL;
END_VAR
VAR_INST
  _bSparse            : Bool;
  _ncount             : uint;
  _eState,
  _eResult            : E_PROGRESS;

  _ndx                : UINT;

  _eProcessState      : E_STATION_STATE;
  _eProcessCmd        : E_STATION_CTRL;

  _nkx                : UINT;

  _nInputLastTarget   : UINT;

{attribute 'displaymode':='bin'}
  _wBufferSentMask    : dword;
{attribute 'displaymode':='bin'}
  _wProcessInputMask  : dWORD; // placement information for movers in stations from preceeding machine
END_VAR
IF NOT Check() THEN AUTO := E_PROGRESS.PROGRESS_ERROR; RETURN; END_IF

//-----------------------------------------------------------------------------
IF NOT Active 
THEN 
	_eState                                     := E_PROGRESS.PROGRESS_INIT;

  _nCount                                     := 0;
  memset(ADR(_nQueue), 0, SIZEOF(_nQueue));
  memset(ADR(_wProcessInputMask), 0, SIZEOF(_wProcessInputMask));
  memset(ADR(_wBufferSentMask), 0, SIZEOF(_wBufferSentMask));
ELSE
  _eProcessState                              := _ItfProcess[_nProcess].ProcessState;

  FOR _ndx := 1 TO MAX_PROCESS
  DO
    _nQueue[_ndx]                             := _ItfProcess[_ndx].MoverCountInQueue;
  END_FOR
END_IF 
//-----------------------------------------------------------------------------
//-----------------------------------------------------------------------------
//-----------------------------------------------------------------------------
CASE _eState
OF
  E_PROGRESS.PROGRESS_INIT:
    IF Active
    THEN
      _nCount := _ncount + 1;
      _wProcessInputMask                      := 0;
      _wBufferSentMask                        := 0;
      _eState                                 := E_PROGRESS.PROGRESS_BUSY;
    END_IF
END_CASE
//-----------------------------------------------------------------------------
//-----------------------------------------------------------------------------
CASE _eState
OF
  E_PROGRESS.PROGRESS_BUSY:

    CASE _nProcess
    OF
      DISTRIBUTOR_2,
      DISTRIBUTOR_1:
        _eState                               := E_PROGRESS.PROGRESS_PREPARE;

      OUTPUT_R2:
        _eState                               := E_PROGRESS.PROGRESS_PREPARE;

      OUTPUT_R1:
        _eState                               := E_PROGRESS.PROGRESS_PREPARE;

      BUFFER_3:
        IF (_nQueue[BUFFER_3] > QUEUE_COUNT)
        THEN
          _eState                             := E_PROGRESS.PROGRESS_PREPARE;
        END_IF

      OUTPUT_1:
        _eState                               := E_PROGRESS.PROGRESS_PREPARE;

      INPUT:
        _eState                               := E_PROGRESS.PROGRESS_PREPARE;

      BUFFER_1:
        _eState                               := E_PROGRESS.PROGRESS_PREPARE;
        IF NOT _bSparse
        THEN
          FOR _nkx := 1 TO _ItfProcess[INPUT].StationCount
          DO
              _wProcessInputMask              := Tc2_System.SETBIT32(_wProcessInputMask, TO_SINT(_nkx-1));
          END_FOR
        ELSE
          FOR _nkx := 1 TO _ItfProcess[INPUT].StationCount
          DO
            IF (_nkx <> 7)
            THEN
              _wProcessInputMask              := _ItfProcess[BUFFER_1].SetBitDWord(_wProcessInputMask, _nkx-1);
            END_IF
          END_FOR

        END_IF


